Yaskawa INFORM job: aprem2TRJ1.JBI

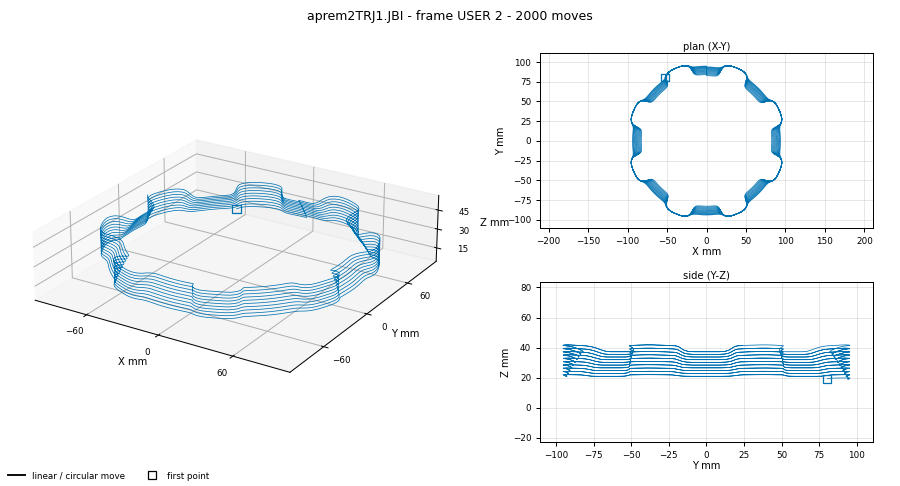
[picture p0: tool path of aprem2TRJ1.JBI in frame USER 2, 2000 of 2000 moves have a stored position in this frame; points joined in program order, loops and branches not executed]
/JOB
//NAME aprem2TRJ1
//POS
///NPOS 2000,0,2000,0,0,0
///USER 2
///TOOL 1
///POSTYPE USER
///RECTAN
///RCONF 1,0,0,0,0,0,0,0,0,0,0,0,0,0,0,0,0,0,0,0,0,0,0,0
C00000=-52.755,80.388,19.309,-171.7434,14.7955,0.0000
C00001=-51.961,81.931,19.493,-175.4363,10.0997,0.0000
C00002=-51.163,83.502,19.627,-176.4604,6.1368,0.0000
C00003=-49.917,85.194,19.692,-177.1673,3.1412,0.0000
C00004=-47.874,87.106,19.726,-178.6253,1.1228,0.0000
C00005=-45.272,88.975,19.753,-179.7684,0.1462,0.0000
C00006=-42.449,90.515,19.780,-179.9313,0.0331,0.0000
C00007=-39.659,91.796,19.798,-179.9923,0.0034,0.0000
C00008=-36.867,92.953,19.798,-179.9922,0.0031,0.0000
C00009=-33.988,94.020,19.780,-179.9280,0.0252,0.0000
C00010=-30.903,94.927,19.753,-179.7329,0.0604,0.0000
C00011=-27.741,95.446,19.726,-178.2343,0.1783,0.0000
C00012=-24.945,95.538,19.692,-175.7796,-0.2187,0.0000
C00013=-22.867,95.222,19.627,-173.1704,-1.8493,0.0000
C00014=-21.192,94.676,19.493,-169.6633,-3.9762,0.0000
C00015=-19.540,94.146,19.309,-163.8609,-4.8105,0.0000
C00016=-17.528,93.824,19.120,-157.6135,-2.4711,0.0000
C00017=-14.592,93.857,18.976,-154.0584,1.6115,0.0000
C00018=-10.190,94.262,18.917,-153.0799,2.7335,0.0000
C00019=-5.317,94.652,18.914,-152.9496,1.6756,0.0000
C00020=0.000,94.804,18.916,-152.9230,0.0002,0.0000
C00021=0.000,93.772,20.859,-151.1709,0.0003,0.0000
C00022=5.223,93.624,20.857,-151.1986,-1.7982,0.0000
C00023=10.031,93.243,20.860,-151.3318,-2.8339,0.0000
C00024=14.399,92.874,20.935,-152.4025,-1.1034,0.0000
C00025=17.292,92.935,21.118,-156.8210,4.1648,0.0000
C00026=19.271,93.399,21.361,-164.4264,6.3648,0.0000
C00027=20.902,94.108,21.598,-170.7334,4.7910,0.0000
C00028=22.556,94.852,21.773,-173.9772,2.3273,0.0000
C00029=24.607,95.353,21.858,-176.1452,0.4720,0.0000
C00030=27.423,95.407,21.902,-178.4246,-0.0969,0.0000
C00031=30.651,94.973,21.938,-179.8436,-0.0322,0.0000
C00032=33.828,94.073,21.973,-179.9356,-0.0223,0.0000
C00033=36.813,92.974,21.997,-179.9932,-0.0027,0.0000
C00034=39.712,91.773,21.997,-179.9933,-0.0029,0.0000
C00035=42.599,90.440,21.973,-179.9387,-0.0298,0.0000
C00036=45.483,88.829,21.938,-179.8667,-0.0878,0.0000
C00037=48.072,86.854,21.902,-178.8174,-1.0456,0.0000
C00038=50.025,84.825,21.858,-177.6053,-3.0607,0.0000
C00039=51.121,83.020,21.773,-177.3739,-5.9001,0.0000
C00040=51.765,81.324,21.598,-176.7889,-9.9060,0.0000
C00041=52.416,79.670,21.361,-173.2589,-15.4269,0.0000
C00042=53.488,77.942,21.118,-165.8953,-19.5067,0.0000
C00043=55.491,75.854,20.935,-159.0309,-19.5961,0.0000
C00044=58.840,73.026,20.860,-157.1386,-19.3725,0.0000
C00045=62.509,69.895,20.857,-157.6594,-20.1308,0.0000
C00046=66.307,66.307,20.859,-158.7340,-21.2663,0.0000
C00047=69.895,62.509,20.857,-159.8689,-22.3404,0.0000
C00048=73.026,58.840,20.860,-160.6271,-22.8610,0.0000
C00049=75.854,55.491,20.935,-160.4041,-20.9693,0.0000
C00050=77.942,53.488,21.118,-160.4933,-14.1047,0.0000
C00051=79.670,52.416,21.361,-164.5731,-6.7411,0.0000
C00052=81.324,51.765,21.598,-170.0940,-3.2111,0.0000
C00053=83.020,51.121,21.773,-174.0999,-2.6261,0.0000
C00054=84.825,50.025,21.858,-176.9393,-2.3947,0.0000
C00055=86.854,48.072,21.902,-178.9544,-1.1826,0.0000
C00056=88.829,45.483,21.938,-179.9122,-0.1333,0.0000
C00057=90.440,42.599,21.973,-179.9702,-0.0613,0.0000
C00058=91.773,39.712,21.997,-179.9971,-0.0067,0.0000
C00059=92.974,36.813,21.997,-179.9973,-0.0068,0.0000
C00060=94.073,33.828,21.973,-179.9777,-0.0644,0.0000
C00061=94.973,30.651,21.938,-179.9678,-0.1564,0.0000
C00062=95.407,27.423,21.902,-179.9031,-1.5754,0.0000
C00063=95.353,24.607,21.858,179.5280,-3.8548,0.0000
C00064=94.852,22.556,21.773,177.6727,-6.0228,0.0000
C00065=94.108,20.902,21.598,175.2090,-9.2666,0.0000
C00066=93.399,19.271,21.361,173.6352,-15.5736,0.0000
C00067=92.935,17.292,21.118,175.8352,-23.1790,0.0000
C00068=92.874,14.399,20.935,-178.8966,-27.5975,0.0000
C00069=93.243,10.031,20.860,-177.1661,-28.6682,0.0000
C00070=93.624,5.223,20.857,-178.2018,-28.8014,0.0000
C00071=93.772,0.000,20.859,179.9997,-28.8291,0.0000
C00072=93.624,-5.223,20.857,178.2021,-28.8014,0.0000
C00073=93.243,-10.031,20.860,177.1667,-28.6682,0.0000
C00074=92.875,-14.399,20.935,178.8963,-27.5974,0.0000
C00075=92.935,-17.292,21.118,-175.8352,-23.1790,0.0000
C00076=93.399,-19.271,21.361,-173.6352,-15.5736,0.0000
C00077=94.108,-20.902,21.598,-175.2090,-9.2666,0.0000
C00078=94.852,-22.556,21.773,-177.6727,-6.0228,0.0000
C00079=95.353,-24.607,21.858,-179.5280,-3.8548,0.0000
C00080=95.407,-27.423,21.902,179.9031,-1.5754,0.0000
C00081=94.973,-30.651,21.938,179.9678,-0.1564,0.0000
C00082=94.073,-33.828,21.973,179.9777,-0.0644,0.0000
C00083=92.974,-36.813,21.997,179.9973,-0.0068,0.0000
C00084=91.773,-39.712,21.997,179.9971,-0.0067,0.0000
C00085=90.440,-42.599,21.973,179.9702,-0.0613,0.0000
C00086=88.829,-45.483,21.938,179.9122,-0.1333,0.0000
C00087=86.854,-48.072,21.902,178.9544,-1.1826,0.0000
C00088=84.825,-50.025,21.858,176.9393,-2.3947,0.0000
C00089=83.020,-51.121,21.773,174.0999,-2.6261,0.0000
C00090=81.324,-51.765,21.598,170.0940,-3.2111,0.0000
C00091=79.670,-52.416,21.361,164.5731,-6.7411,0.0000
C00092=77.942,-53.488,21.118,160.4933,-14.1047,0.0000
C00093=75.854,-55.491,20.935,160.4039,-20.9691,0.0000
C00094=73.026,-58.840,20.860,160.6275,-22.8614,0.0000
C00095=69.895,-62.509,20.857,159.8692,-22.3406,0.0000
C00096=66.307,-66.307,20.859,158.7337,-21.2660,0.0000
C00097=62.509,-69.895,20.857,157.6596,-20.1311,0.0000
C00098=58.840,-73.026,20.860,157.1390,-19.3729,0.0000
C00099=55.491,-75.854,20.935,159.0307,-19.5959,0.0000
C00100=53.488,-77.942,21.118,165.8953,-19.5067,0.0000
C00101=52.416,-79.670,21.361,173.2589,-15.4269,0.0000
C00102=51.765,-81.324,21.598,176.7889,-9.9060,0.0000
C00103=51.121,-83.020,21.773,177.3739,-5.9001,0.0000
C00104=50.025,-84.825,21.858,177.6053,-3.0607,0.0000
C00105=48.072,-86.854,21.902,178.8174,-1.0456,0.0000
C00106=45.483,-88.829,21.938,179.8667,-0.0878,0.0000
C00107=42.599,-90.440,21.973,179.9387,-0.0298,0.0000
C00108=39.712,-91.773,21.997,179.9933,-0.0029,0.0000
C00109=36.813,-92.974,21.997,179.9932,-0.0027,0.0000
C00110=33.828,-94.073,21.973,179.9356,-0.0223,0.0000
C00111=30.651,-94.973,21.938,179.8436,-0.0322,0.0000
C00112=27.423,-95.407,21.902,178.4246,-0.0969,0.0000
C00113=24.607,-95.353,21.858,176.1452,0.4720,0.0000
C00114=22.556,-94.852,21.773,173.9772,2.3273,0.0000
C00115=20.902,-94.108,21.598,170.7334,4.7910,0.0000
C00116=19.271,-93.399,21.361,164.4264,6.3648,0.0000
C00117=17.292,-92.935,21.118,156.8210,4.1648,0.0000
C00118=14.399,-92.874,20.935,152.4025,-1.1034,0.0000
C00119=10.031,-93.243,20.860,151.3318,-2.8339,0.0000
C00120=5.223,-93.624,20.857,151.1986,-1.7982,0.0000
C00121=0.000,-93.772,20.859,151.1709,0.0003,0.0000
C00122=0.000,-93.772,20.859,151.1709,0.0003,0.0000
C00123=-5.223,-93.624,20.857,151.1986,1.7979,0.0000
C00124=-10.031,-93.243,20.860,151.3318,2.8333,0.0000
C00125=-14.399,-92.875,20.935,152.4026,1.1037,0.0000
C00126=-17.292,-92.935,21.118,156.8210,-4.1648,0.0000
C00127=-19.271,-93.399,21.361,164.4264,-6.3648,0.0000
C00128=-20.902,-94.108,21.598,170.7334,-4.7910,0.0000
C00129=-22.556,-94.852,21.773,173.9772,-2.3273,0.0000
C00130=-24.607,-95.353,21.858,176.1452,-0.4720,0.0000
C00131=-27.423,-95.407,21.902,178.4246,0.0969,0.0000
C00132=-30.651,-94.973,21.938,179.8436,0.0322,0.0000
C00133=-33.828,-94.073,21.973,179.9356,0.0223,0.0000
C00134=-36.813,-92.974,21.997,179.9932,0.0027,0.0000
C00135=-39.712,-91.773,21.997,179.9933,0.0029,0.0000
C00136=-42.599,-90.440,21.973,179.9387,0.0298,0.0000
C00137=-45.483,-88.829,21.938,179.8667,0.0878,0.0000
C00138=-48.072,-86.854,21.902,178.8174,1.0456,0.0000
C00139=-50.025,-84.825,21.858,177.6053,3.0607,0.0000
C00140=-51.121,-83.020,21.773,177.3739,5.9001,0.0000
C00141=-51.765,-81.324,21.598,176.7889,9.9060,0.0000
C00142=-52.416,-79.670,21.361,173.2589,15.4269,0.0000
C00143=-53.488,-77.942,21.118,165.8953,19.5067,0.0000
C00144=-55.491,-75.854,20.935,159.0309,19.5961,0.0000
C00145=-58.840,-73.026,20.860,157.1386,19.3725,0.0000
C00146=-62.509,-69.895,20.857,157.6594,20.1308,0.0000
C00147=-66.307,-66.307,20.859,158.7340,21.2663,0.0000
C00148=-69.895,-62.509,20.857,159.8689,22.3404,0.0000
C00149=-73.026,-58.840,20.860,160.6271,22.8610,0.0000
C00150=-75.854,-55.491,20.935,160.4041,20.9693,0.0000
C00151=-77.942,-53.488,21.118,160.4933,14.1047,0.0000
C00152=-79.670,-52.416,21.361,164.5731,6.7411,0.0000
C00153=-81.324,-51.765,21.598,170.0940,3.2111,0.0000
C00154=-83.020,-51.121,21.773,174.0999,2.6261,0.0000
C00155=-84.825,-50.025,21.858,176.9393,2.3947,0.0000
C00156=-86.854,-48.072,21.902,178.9544,1.1826,0.0000
C00157=-88.829,-45.483,21.938,179.9122,0.1333,0.0000
C00158=-90.440,-42.599,21.973,179.9702,0.0613,0.0000
C00159=-91.773,-39.712,21.997,179.9971,0.0067,0.0000
C00160=-92.974,-36.813,21.997,179.9973,0.0068,0.0000
C00161=-94.073,-33.828,21.973,179.9777,0.0644,0.0000
C00162=-94.973,-30.651,21.938,179.9678,0.1564,0.0000
C00163=-95.407,-27.423,21.902,179.9031,1.5754,0.0000
C00164=-95.353,-24.607,21.858,-179.5280,3.8548,0.0000
C00165=-94.852,-22.556,21.773,-177.6727,6.0228,0.0000
C00166=-94.108,-20.902,21.598,-175.2090,9.2666,0.0000
C00167=-93.399,-19.271,21.361,-173.6352,15.5736,0.0000
C00168=-92.935,-17.292,21.118,-175.8352,23.1790,0.0000
C00169=-92.874,-14.399,20.935,178.8966,27.5975,0.0000
C00170=-93.243,-10.031,20.860,177.1661,28.6682,0.0000
C00171=-93.624,-5.223,20.857,178.2018,28.8014,0.0000
C00172=-93.772,0.000,20.859,-179.9997,28.8291,0.0000
C00173=-93.624,5.223,20.857,-178.2021,28.8014,0.0000
C00174=-93.243,10.031,20.860,-177.1667,28.6682,0.0000
C00175=-92.875,14.399,20.935,-178.8963,27.5974,0.0000
C00176=-92.935,17.292,21.118,175.8352,23.1790,0.0000
C00177=-93.399,19.271,21.361,173.6352,15.5736,0.0000
C00178=-94.108,20.902,21.598,175.2090,9.2666,0.0000
C00179=-94.852,22.556,21.773,177.6727,6.0228,0.0000
C00180=-95.353,24.607,21.858,179.5280,3.8548,0.0000
C00181=-95.407,27.423,21.902,-179.9031,1.5754,0.0000
C00182=-94.973,30.651,21.938,-179.9678,0.1564,0.0000
C00183=-94.073,33.828,21.973,-179.9777,0.0644,0.0000
C00184=-92.974,36.813,21.997,-179.9973,0.0068,0.0000
C00185=-91.773,39.712,21.997,-179.9971,0.0067,0.0000
C00186=-90.440,42.599,21.973,-179.9702,0.0613,0.0000
C00187=-88.829,45.483,21.938,-179.9122,0.1333,0.0000
C00188=-86.854,48.072,21.902,-178.9544,1.1826,0.0000
C00189=-84.825,50.025,21.858,-176.9393,2.3947,0.0000
C00190=-83.020,51.121,21.773,-174.0999,2.6261,0.0000
C00191=-81.324,51.765,21.598,-170.0940,3.2111,0.0000
C00192=-79.670,52.416,21.361,-164.5731,6.7411,0.0000
C00193=-77.942,53.488,21.118,-160.4933,14.1047,0.0000
C00194=-75.854,55.491,20.935,-160.4039,20.9691,0.0000
C00195=-73.026,58.840,20.860,-160.6275,22.8614,0.0000
C00196=-69.895,62.509,20.857,-159.8692,22.3406,0.0000
C00197=-66.307,66.307,20.859,-158.7337,21.2660,0.0000
C00198=-62.509,69.895,20.857,-157.6596,20.1311,0.0000
C00199=-58.840,73.026,20.860,-157.1390,19.3729,0.0000
C00200=-55.491,75.854,20.935,-159.0307,19.5959,0.0000
C00201=-53.488,77.942,21.118,-165.8953,19.5067,0.0000
C00202=-52.416,79.670,21.361,-173.2589,15.4269,0.0000
C00203=-51.765,81.324,21.598,-176.7889,9.9060,0.0000
C00204=-51.121,83.020,21.773,-177.3739,5.9001,0.0000
C00205=-50.025,84.825,21.858,-177.6053,3.0607,0.0000
C00206=-48.072,86.854,21.902,-178.8174,1.0456,0.0000
C00207=-45.483,88.829,21.938,-179.8667,0.0878,0.0000
C00208=-42.599,90.440,21.973,-179.9387,0.0298,0.0000
C00209=-39.712,91.773,21.997,-179.9933,0.0029,0.0000
C00210=-36.813,92.974,21.997,-179.9932,0.0027,0.0000
C00211=-33.828,94.073,21.973,-179.9356,0.0223,0.0000
C00212=-30.651,94.973,21.938,-179.8436,0.0322,0.0000
C00213=-27.423,95.407,21.902,-178.4246,0.0969,0.0000
C00214=-24.607,95.353,21.858,-176.1452,-0.4720,0.0000
C00215=-22.556,94.852,21.773,-173.9772,-2.3273,0.0000
C00216=-20.902,94.108,21.598,-170.7334,-4.7910,0.0000
C00217=-19.271,93.399,21.361,-164.4264,-6.3648,0.0000
C00218=-17.292,92.935,21.118,-156.8210,-4.1648,0.0000
C00219=-14.399,92.875,20.935,-152.4026,1.1037,0.0000
C00220=-10.031,93.243,20.860,-151.3318,2.8333,0.0000
C00221=-5.223,93.624,20.857,-151.1986,1.7979,0.0000
C00222=0.000,93.772,20.859,-151.1709,0.0003,0.0000
C00223=0.000,92.684,22.771,-149.6099,0.0003,0.0000
C00224=5.124,92.540,22.769,-149.6384,-1.9089,0.0000
C00225=9.864,92.169,22.773,-149.7740,-2.8935,0.0000
C00226=14.194,91.838,22.865,-150.9609,-0.4562,0.0000
C00227=17.042,91.994,23.091,-156.4950,5.9927,0.0000
C00228=18.986,92.606,23.393,-165.5257,7.6266,0.0000
C00229=20.592,93.503,23.691,-172.1237,5.1935,0.0000
C00230=22.223,94.456,23.912,-175.0607,2.5303,0.0000
C00231=24.245,95.156,24.019,-176.7061,0.6541,0.0000
C00232=27.082,95.366,24.075,-178.6926,-0.0269,0.0000
C00233=30.380,95.022,24.120,-179.9786,-0.0040,0.0000
C00234=33.658,94.129,24.166,-179.9455,-0.0187,0.0000
C00235=36.755,92.996,24.196,-179.9945,-0.0022,0.0000
C00236=39.769,91.748,24.196,-179.9946,-0.0024,0.0000
C00237=42.760,90.359,24.166,-179.9482,-0.0253,0.0000
C00238=45.709,88.673,24.120,-179.9821,-0.0123,0.0000
C00239=48.284,86.584,24.075,-179.0565,-0.9056,0.0000
C00240=50.142,84.429,24.019,-178.1315,-2.7920,0.0000
C00241=51.076,82.504,23.912,-178.2896,-5.2767,0.0000
C00242=51.556,80.678,23.691,-178.0785,-9.2071,0.0000
C00243=52.057,78.907,23.393,-174.9794,-15.4942,0.0000
C00244=52.999,77.101,23.091,-166.8676,-20.8949,0.0000
C00245=54.903,74.976,22.865,-158.2868,-21.1542,0.0000
C00246=58.198,72.148,22.773,-155.8812,-20.6181,0.0000
C00247=61.813,69.059,22.769,-156.3569,-21.3383,0.0000
C00248=65.538,65.538,22.771,-157.4767,-22.5237,0.0000
C00249=69.059,61.813,22.769,-158.6615,-23.6429,0.0000
C00250=72.148,58.198,22.773,-159.3815,-24.1184,0.0000
C00251=74.976,54.903,22.865,-158.8460,-21.7135,0.0000
C00252=77.101,52.999,23.091,-159.1051,-13.1324,0.0000
C00253=78.907,52.057,23.393,-164.5058,-5.0206,0.0000
C00254=80.678,51.556,23.691,-170.7929,-1.9215,0.0000
C00255=82.504,51.076,23.912,-174.7233,-1.7104,0.0000
C00256=84.429,50.142,24.019,-177.2080,-1.8685,0.0000
C00257=86.584,48.284,24.075,-179.0944,-0.9435,0.0000
C00258=88.673,45.709,24.120,-179.9877,-0.0179,0.0000
C00259=90.359,42.760,24.166,-179.9747,-0.0518,0.0000
C00260=91.748,39.769,24.196,-179.9976,-0.0054,0.0000
C00261=92.996,36.755,24.196,-179.9978,-0.0055,0.0000
C00262=94.129,33.658,24.166,-179.9813,-0.0545,0.0000
C00263=95.022,30.380,24.120,-179.9960,-0.0214,0.0000
C00264=95.366,27.082,24.075,-179.9731,-1.3074,0.0000
C00265=95.156,24.245,24.019,179.3459,-3.2939,0.0000
C00266=94.456,22.223,23.912,177.4697,-4.9393,0.0000
C00267=93.503,20.592,23.691,174.8065,-7.8763,0.0000
C00268=92.606,18.986,23.393,172.3734,-14.4743,0.0000
C00269=91.994,17.042,23.091,174.0073,-23.5050,0.0000
C00270=91.838,14.194,22.865,-179.5438,-29.0391,0.0000
C00271=92.169,9.864,22.773,-177.1065,-30.2260,0.0000
C00272=92.540,5.124,22.769,-178.0911,-30.3616,0.0000
C00273=92.684,0.000,22.771,179.9997,-30.3901,0.0000
C00274=92.540,-5.124,22.769,178.0916,-30.3616,0.0000
C00275=92.169,-9.864,22.773,177.1071,-30.2260,0.0000
C00276=91.838,-14.194,22.865,179.5434,-29.0390,0.0000
C00277=91.994,-17.042,23.091,-174.0073,-23.5050,0.0000
C00278=92.606,-18.986,23.393,-172.3734,-14.4743,0.0000
C00279=93.503,-20.592,23.691,-174.8065,-7.8763,0.0000
C00280=94.456,-22.223,23.912,-177.4697,-4.9393,0.0000
C00281=95.156,-24.245,24.019,-179.3459,-3.2939,0.0000
C00282=95.366,-27.082,24.075,179.9731,-1.3074,0.0000
C00283=95.022,-30.380,24.120,179.9960,-0.0214,0.0000
C00284=94.129,-33.658,24.166,179.9813,-0.0545,0.0000
C00285=92.996,-36.755,24.196,179.9978,-0.0055,0.0000
C00286=91.748,-39.769,24.196,179.9976,-0.0054,0.0000
C00287=90.359,-42.760,24.166,179.9747,-0.0518,0.0000
C00288=88.673,-45.709,24.120,179.9877,-0.0179,0.0000
C00289=86.584,-48.284,24.075,179.0944,-0.9435,0.0000
C00290=84.429,-50.142,24.019,177.2080,-1.8685,0.0000
C00291=82.504,-51.076,23.912,174.7233,-1.7104,0.0000
C00292=80.678,-51.556,23.691,170.7929,-1.9215,0.0000
C00293=78.907,-52.057,23.393,164.5058,-5.0206,0.0000
C00294=77.101,-52.999,23.091,159.1051,-13.1324,0.0000
C00295=74.976,-54.903,22.865,158.8458,-21.7132,0.0000
C00296=72.148,-58.198,22.773,159.3819,-24.1188,0.0000
C00297=69.059,-61.813,22.769,158.6617,-23.6431,0.0000
C00298=65.538,-65.538,22.771,157.4763,-22.5233,0.0000
C00299=61.813,-69.059,22.769,156.3571,-21.3385,0.0000
C00300=58.198,-72.148,22.773,155.8816,-20.6185,0.0000
C00301=54.903,-74.976,22.865,158.2865,-21.1540,0.0000
C00302=52.999,-77.101,23.091,166.8676,-20.8949,0.0000
C00303=52.057,-78.907,23.393,174.9794,-15.4942,0.0000
C00304=51.556,-80.678,23.691,178.0785,-9.2071,0.0000
C00305=51.076,-82.504,23.912,178.2896,-5.2767,0.0000
C00306=50.142,-84.429,24.019,178.1315,-2.7920,0.0000
C00307=48.284,-86.584,24.075,179.0565,-0.9056,0.0000
C00308=45.709,-88.673,24.120,179.9821,-0.0123,0.0000
C00309=42.760,-90.359,24.166,179.9482,-0.0253,0.0000
C00310=39.769,-91.748,24.196,179.9946,-0.0024,0.0000
C00311=36.755,-92.996,24.196,179.9945,-0.0022,0.0000
C00312=33.658,-94.129,24.166,179.9455,-0.0187,0.0000
C00313=30.380,-95.022,24.120,179.9786,-0.0040,0.0000
C00314=27.082,-95.366,24.075,178.6926,-0.0269,0.0000
C00315=24.245,-95.156,24.019,176.7061,0.6541,0.0000
C00316=22.223,-94.456,23.912,175.0607,2.5303,0.0000
C00317=20.592,-93.503,23.691,172.1237,5.1935,0.0000
C00318=18.986,-92.606,23.393,165.5257,7.6266,0.0000
C00319=17.042,-91.994,23.091,156.4950,5.9927,0.0000
C00320=14.194,-91.838,22.865,150.9609,-0.4562,0.0000
C00321=9.864,-92.169,22.773,149.7740,-2.8935,0.0000
C00322=5.124,-92.540,22.769,149.6384,-1.9089,0.0000
C00323=0.000,-92.684,22.771,149.6099,0.0003,0.0000
C00324=0.000,-92.684,22.771,149.6099,0.0003,0.0000
C00325=-5.124,-92.540,22.769,149.6384,1.9084,0.0000
C00326=-9.864,-92.169,22.773,149.7740,2.8929,0.0000
C00327=-14.194,-91.838,22.865,150.9610,0.4566,0.0000
C00328=-17.042,-91.994,23.091,156.4950,-5.9927,0.0000
C00329=-18.986,-92.606,23.393,165.5257,-7.6266,0.0000
C00330=-20.592,-93.503,23.691,172.1237,-5.1935,0.0000
C00331=-22.223,-94.456,23.912,175.0607,-2.5303,0.0000
C00332=-24.245,-95.156,24.019,176.7061,-0.6541,0.0000
C00333=-27.082,-95.366,24.075,178.6926,0.0269,0.0000
C00334=-30.380,-95.022,24.120,179.9786,0.0040,0.0000
C00335=-33.658,-94.129,24.166,179.9455,0.0187,0.0000
C00336=-36.755,-92.996,24.196,179.9945,0.0022,0.0000
C00337=-39.769,-91.748,24.196,179.9946,0.0024,0.0000
C00338=-42.760,-90.359,24.166,179.9482,0.0253,0.0000
C00339=-45.709,-88.673,24.120,179.9821,0.0123,0.0000
C00340=-48.284,-86.584,24.075,179.0565,0.9056,0.0000
C00341=-50.142,-84.429,24.019,178.1315,2.7920,0.0000
C00342=-51.076,-82.504,23.912,178.2896,5.2767,0.0000
C00343=-51.556,-80.678,23.691,178.0785,9.2071,0.0000
C00344=-52.057,-78.907,23.393,174.9794,15.4942,0.0000
C00345=-52.999,-77.101,23.091,166.8676,20.8949,0.0000
C00346=-54.903,-74.976,22.865,158.2868,21.1542,0.0000
C00347=-58.198,-72.148,22.773,155.8812,20.6181,0.0000
C00348=-61.813,-69.059,22.769,156.3569,21.3383,0.0000
C00349=-65.538,-65.538,22.771,157.4767,22.5237,0.0000
C00350=-69.059,-61.813,22.769,158.6615,23.6429,0.0000
C00351=-72.148,-58.198,22.773,159.3815,24.1184,0.0000
C00352=-74.976,-54.903,22.865,158.8460,21.7135,0.0000
C00353=-77.101,-52.999,23.091,159.1051,13.1324,0.0000
C00354=-78.907,-52.057,23.393,164.5058,5.0206,0.0000
C00355=-80.678,-51.556,23.691,170.7929,1.9215,0.0000
C00356=-82.504,-51.076,23.912,174.7233,1.7104,0.0000
C00357=-84.429,-50.142,24.019,177.2080,1.8685,0.0000
C00358=-86.584,-48.284,24.075,179.0944,0.9435,0.0000
C00359=-88.673,-45.709,24.120,179.9877,0.0179,0.0000
C00360=-90.359,-42.760,24.166,179.9747,0.0518,0.0000
C00361=-91.748,-39.769,24.196,179.9976,0.0054,0.0000
C00362=-92.996,-36.755,24.196,179.9978,0.0055,0.0000
C00363=-94.129,-33.658,24.166,179.9813,0.0545,0.0000
C00364=-95.022,-30.380,24.120,179.9960,0.0214,0.0000
C00365=-95.366,-27.082,24.075,179.9731,1.3074,0.0000
C00366=-95.156,-24.245,24.019,-179.3459,3.2939,0.0000
C00367=-94.456,-22.223,23.912,-177.4697,4.9393,0.0000
C00368=-93.503,-20.592,23.691,-174.8065,7.8763,0.0000
C00369=-92.606,-18.986,23.393,-172.3734,14.4743,0.0000
C00370=-91.994,-17.042,23.091,-174.0073,23.5050,0.0000
C00371=-91.838,-14.194,22.865,179.5438,29.0391,0.0000
C00372=-92.169,-9.864,22.773,177.1065,30.2260,0.0000
C00373=-92.540,-5.124,22.769,178.0911,30.3616,0.0000
C00374=-92.684,0.000,22.771,-179.9997,30.3901,0.0000
C00375=-92.540,5.124,22.769,-178.0916,30.3616,0.0000
C00376=-92.169,9.864,22.773,-177.1071,30.2260,0.0000
C00377=-91.838,14.194,22.865,-179.5434,29.0390,0.0000
C00378=-91.994,17.042,23.091,174.0073,23.5050,0.0000
C00379=-92.606,18.986,23.393,172.3734,14.4743,0.0000
C00380=-93.503,20.592,23.691,174.8065,7.8763,0.0000
C00381=-94.456,22.223,23.912,177.4697,4.9393,0.0000
C00382=-95.156,24.245,24.019,179.3459,3.2939,0.0000
C00383=-95.366,27.082,24.075,-179.9731,1.3074,0.0000
C00384=-95.022,30.380,24.120,-179.9960,0.0214,0.0000
C00385=-94.129,33.658,24.166,-179.9813,0.0545,0.0000
C00386=-92.996,36.755,24.196,-179.9978,0.0055,0.0000
C00387=-91.748,39.769,24.196,-179.9976,0.0054,0.0000
C00388=-90.359,42.760,24.166,-179.9747,0.0518,0.0000
C00389=-88.673,45.709,24.120,-179.9877,0.0179,0.0000
C00390=-86.584,48.284,24.075,-179.0944,0.9435,0.0000
C00391=-84.429,50.142,24.019,-177.2080,1.8685,0.0000
C00392=-82.504,51.076,23.912,-174.7233,1.7104,0.0000
C00393=-80.678,51.556,23.691,-170.7929,1.9215,0.0000
C00394=-78.907,52.057,23.393,-164.5058,5.0206,0.0000
C00395=-77.101,52.999,23.091,-159.1051,13.1324,0.0000
C00396=-74.976,54.903,22.865,-158.8458,21.7132,0.0000
C00397=-72.148,58.198,22.773,-159.3819,24.1188,0.0000
C00398=-69.059,61.813,22.769,-158.6617,23.6431,0.0000
C00399=-65.538,65.538,22.771,-157.4763,22.5233,0.0000
C00400=-61.813,69.059,22.769,-156.3571,21.3385,0.0000
C00401=-58.198,72.148,22.773,-155.8816,20.6185,0.0000
C00402=-54.903,74.976,22.865,-158.2865,21.1540,0.0000
C00403=-52.999,77.101,23.091,-166.8676,20.8949,0.0000
C00404=-52.057,78.907,23.393,-174.9794,15.4942,0.0000
C00405=-51.556,80.678,23.691,-178.0785,9.2071,0.0000
C00406=-51.076,82.504,23.912,-178.2896,5.2767,0.0000
C00407=-50.142,84.429,24.019,-178.1315,2.7920,0.0000
C00408=-48.284,86.584,24.075,-179.0565,0.9056,0.0000
C00409=-45.709,88.673,24.120,-179.9821,0.0123,0.0000
C00410=-42.760,90.359,24.166,-179.9482,0.0253,0.0000
C00411=-39.769,91.748,24.196,-179.9946,0.0024,0.0000
C00412=-36.755,92.996,24.196,-179.9945,0.0022,0.0000
C00413=-33.658,94.129,24.166,-179.9455,0.0187,0.0000
C00414=-30.380,95.022,24.120,-179.9786,0.0040,0.0000
C00415=-27.082,95.366,24.075,-178.6926,0.0269,0.0000
C00416=-24.245,95.156,24.019,-176.7061,-0.6541,0.0000
C00417=-22.223,94.456,23.912,-175.0607,-2.5303,0.0000
C00418=-20.592,93.503,23.691,-172.1237,-5.1935,0.0000
C00419=-18.986,92.606,23.393,-165.5257,-7.6266,0.0000
C00420=-17.042,91.994,23.091,-156.4950,-5.9927,0.0000
C00421=-14.194,91.838,22.865,-150.9610,0.4566,0.0000
C00422=-9.864,92.169,22.773,-149.7740,2.8929,0.0000
C00423=-5.124,92.540,22.769,-149.6384,1.9084,0.0000
C00424=0.000,92.684,22.771,-149.6099,0.0003,0.0000
C00425=0.000,91.548,24.655,-148.2220,0.0004,0.0000
C00426=5.020,91.408,24.652,-148.2512,-2.0082,0.0000
C00427=9.690,91.047,24.657,-148.3888,-2.9141,0.0000
C00428=13.981,90.755,24.767,-149.7234,0.3213,0.0000
C00429=16.781,91.008,25.041,-156.6468,7.8344,0.0000
C00430=18.686,91.772,25.406,-167.0189,8.4697,0.0000
C00431=20.265,92.865,25.771,-173.6442,5.1590,0.0000
C00432=21.871,94.037,26.043,-176.2884,2.4064,0.0000
C00433=23.861,94.948,26.175,-177.4309,0.7190,0.0000
C00434=26.720,95.323,26.245,-179.0289,0.0208,0.0000
C00435=30.093,95.074,26.301,179.8658,0.0220,0.0000
C00436=33.476,94.189,26.358,-179.9573,-0.0145,0.0000
C00437=36.693,93.020,26.395,-179.9960,-0.0016,0.0000
C00438=39.829,91.721,26.395,-179.9960,-0.0018,0.0000
C00439=42.931,90.273,26.358,-179.9596,-0.0199,0.0000
C00440=45.948,88.507,26.301,179.8895,0.0793,0.0000
C00441=48.509,86.297,26.245,-179.3280,-0.7014,0.0000
C00442=50.266,84.010,26.175,-178.6908,-2.3250,0.0000
C00443=51.029,81.959,26.043,-179.0745,-4.3225,0.0000
C00444=51.336,79.995,25.771,-179.1451,-8.1159,0.0000
C00445=51.679,78.105,25.406,-176.6973,-15.0186,0.0000
C00446=52.487,76.218,25.041,-168.2493,-21.9298,0.0000
C00447=54.287,74.059,24.767,-157.7629,-22.6253,0.0000
C00448=57.528,71.231,24.657,-154.7702,-21.7624,0.0000
C00449=61.085,68.184,24.652,-155.1868,-22.4287,0.0000
C00450=64.734,64.734,24.655,-156.3444,-23.6560,0.0000
C00451=68.184,61.085,24.652,-157.5710,-24.8129,0.0000
C00452=71.231,57.528,24.657,-158.2372,-25.2293,0.0000
C00453=74.059,54.287,24.767,-157.3750,-22.2374,0.0000
C00454=76.218,52.487,25.041,-158.0702,-11.7507,0.0000
C00455=78.105,51.679,25.406,-164.9814,-3.3027,0.0000
C00456=79.995,51.336,25.771,-171.8841,-0.8549,0.0000
C00457=81.959,51.029,26.043,-175.6775,-0.9255,0.0000
C00458=84.010,50.266,26.175,-177.6750,-1.3092,0.0000
C00459=86.297,48.509,26.245,-179.2986,-0.6720,0.0000
C00460=88.507,45.948,26.301,179.9207,0.1105,0.0000
C00461=90.273,42.931,26.358,-179.9801,-0.0404,0.0000
C00462=91.721,39.829,26.395,-179.9982,-0.0040,0.0000
C00463=93.020,36.693,26.395,-179.9984,-0.0040,0.0000
C00464=94.189,33.476,26.358,-179.9855,-0.0427,0.0000
C00465=95.074,30.093,26.301,179.9780,0.1342,0.0000
C00466=95.323,26.720,26.245,179.9792,-0.9711,0.0000
C00467=94.948,23.861,26.175,179.2810,-2.5691,0.0000
C00468=94.037,21.871,26.043,177.5936,-3.7116,0.0000
C00469=92.865,20.265,25.771,174.8410,-6.3558,0.0000
C00470=91.772,18.686,25.406,171.5303,-12.9811,0.0000
C00471=91.008,16.781,25.041,172.1656,-23.3532,0.0000
C00472=90.755,13.981,24.767,179.6787,-30.2766,0.0000
C00473=91.047,9.690,24.657,-177.0859,-31.6112,0.0000
C00474=91.408,5.020,24.652,-177.9918,-31.7488,0.0000
C00475=91.548,0.000,24.655,179.9996,-31.7780,0.0000
C00476=91.408,-5.020,24.652,177.9923,-31.7488,0.0000
C00477=91.047,-9.690,24.657,177.0867,-31.6111,0.0000
C00478=90.755,-13.981,24.767,-179.6793,-30.2766,0.0000
C00479=91.008,-16.781,25.041,-172.1656,-23.3532,0.0000
C00480=91.772,-18.686,25.406,-171.5303,-12.9811,0.0000
C00481=92.865,-20.265,25.771,-174.8410,-6.3558,0.0000
C00482=94.037,-21.871,26.043,-177.5936,-3.7116,0.0000
C00483=94.948,-23.861,26.175,-179.2810,-2.5691,0.0000
C00484=95.323,-26.720,26.245,-179.9792,-0.9711,0.0000
C00485=95.074,-30.093,26.301,-179.9780,0.1342,0.0000
C00486=94.189,-33.476,26.358,179.9855,-0.0427,0.0000
C00487=93.020,-36.693,26.395,179.9984,-0.0040,0.0000
C00488=91.721,-39.829,26.395,179.9982,-0.0040,0.0000
C00489=90.273,-42.931,26.358,179.9801,-0.0404,0.0000
C00490=88.507,-45.948,26.301,-179.9207,0.1105,0.0000
C00491=86.297,-48.509,26.245,179.2986,-0.6720,0.0000
C00492=84.010,-50.266,26.175,177.6750,-1.3092,0.0000
C00493=81.959,-51.029,26.043,175.6775,-0.9255,0.0000
C00494=79.995,-51.336,25.771,171.8841,-0.8549,0.0000
C00495=78.105,-51.679,25.406,164.9814,-3.3027,0.0000
C00496=76.218,-52.487,25.041,158.0702,-11.7507,0.0000
C00497=74.059,-54.287,24.767,157.3747,-22.2371,0.0000
C00498=71.231,-57.528,24.657,158.2376,-25.2298,0.0000
C00499=68.184,-61.085,24.652,157.5713,-24.8132,0.0000
C00500=64.734,-64.734,24.655,156.3440,-23.6556,0.0000
C00501=61.085,-68.184,24.652,155.1871,-22.4290,0.0000
C00502=57.528,-71.231,24.657,154.7707,-21.7628,0.0000
C00503=54.287,-74.059,24.767,157.7626,-22.6250,0.0000
C00504=52.487,-76.218,25.041,168.2493,-21.9298,0.0000
C00505=51.679,-78.105,25.406,176.6973,-15.0186,0.0000
C00506=51.336,-79.995,25.771,179.1451,-8.1159,0.0000
C00507=51.029,-81.959,26.043,179.0745,-4.3225,0.0000
C00508=50.266,-84.010,26.175,178.6908,-2.3250,0.0000
C00509=48.509,-86.297,26.245,179.3280,-0.7014,0.0000
C00510=45.948,-88.507,26.301,-179.8895,0.0793,0.0000
C00511=42.931,-90.273,26.358,179.9596,-0.0199,0.0000
C00512=39.829,-91.721,26.395,179.9960,-0.0018,0.0000
C00513=36.693,-93.020,26.395,179.9960,-0.0016,0.0000
C00514=33.476,-94.189,26.358,179.9573,-0.0145,0.0000
C00515=30.093,-95.074,26.301,-179.8658,0.0220,0.0000
C00516=26.720,-95.323,26.245,179.0289,0.0208,0.0000
C00517=23.861,-94.948,26.175,177.4309,0.7190,0.0000
C00518=21.871,-94.037,26.043,176.2884,2.4064,0.0000
C00519=20.265,-92.865,25.771,173.6442,5.1590,0.0000
C00520=18.686,-91.772,25.406,167.0189,8.4697,0.0000
C00521=16.781,-91.008,25.041,156.6468,7.8344,0.0000
C00522=13.981,-90.755,24.767,149.7234,0.3213,0.0000
C00523=9.690,-91.047,24.657,148.3888,-2.9141,0.0000
C00524=5.020,-91.408,24.652,148.2512,-2.0082,0.0000
C00525=0.000,-91.548,24.655,148.2220,0.0004,0.0000
C00526=0.000,-91.548,24.655,148.2220,0.0004,0.0000
C00527=-5.020,-91.408,24.652,148.2512,2.0077,0.0000
C00528=-9.690,-91.047,24.657,148.3889,2.9133,0.0000
C00529=-13.981,-90.755,24.767,149.7234,-0.3207,0.0000
C00530=-16.781,-91.008,25.041,156.6468,-7.8344,0.0000
C00531=-18.686,-91.772,25.406,167.0189,-8.4697,0.0000
C00532=-20.265,-92.865,25.771,173.6442,-5.1590,0.0000
C00533=-21.871,-94.037,26.043,176.2884,-2.4064,0.0000
C00534=-23.861,-94.948,26.175,177.4309,-0.7190,0.0000
C00535=-26.720,-95.323,26.245,179.0289,-0.0208,0.0000
C00536=-30.093,-95.074,26.301,-179.8658,-0.0220,0.0000
C00537=-33.476,-94.189,26.358,179.9573,0.0145,0.0000
C00538=-36.693,-93.020,26.395,179.9960,0.0016,0.0000
C00539=-39.829,-91.721,26.395,179.9960,0.0018,0.0000
C00540=-42.931,-90.273,26.358,179.9596,0.0199,0.0000
C00541=-45.948,-88.507,26.301,-179.8895,-0.0793,0.0000
C00542=-48.509,-86.297,26.245,179.3280,0.7014,0.0000
C00543=-50.266,-84.010,26.175,178.6908,2.3250,0.0000
C00544=-51.029,-81.959,26.043,179.0745,4.3225,0.0000
C00545=-51.336,-79.995,25.771,179.1451,8.1159,0.0000
C00546=-51.679,-78.105,25.406,176.6973,15.0186,0.0000
C00547=-52.487,-76.218,25.041,168.2493,21.9298,0.0000
C00548=-54.287,-74.059,24.767,157.7629,22.6253,0.0000
C00549=-57.528,-71.231,24.657,154.7702,21.7624,0.0000
C00550=-61.085,-68.184,24.652,155.1868,22.4287,0.0000
C00551=-64.734,-64.734,24.655,156.3444,23.6560,0.0000
C00552=-68.184,-61.085,24.652,157.5710,24.8129,0.0000
C00553=-71.231,-57.528,24.657,158.2372,25.2293,0.0000
C00554=-74.059,-54.287,24.767,157.3750,22.2374,0.0000
C00555=-76.218,-52.487,25.041,158.0702,11.7507,0.0000
C00556=-78.105,-51.679,25.406,164.9814,3.3027,0.0000
C00557=-79.995,-51.336,25.771,171.8841,0.8549,0.0000
C00558=-81.959,-51.029,26.043,175.6775,0.9255,0.0000
C00559=-84.010,-50.266,26.175,177.6750,1.3092,0.0000
C00560=-86.297,-48.509,26.245,179.2986,0.6720,0.0000
C00561=-88.507,-45.948,26.301,-179.9207,-0.1105,0.0000
C00562=-90.273,-42.931,26.358,179.9801,0.0404,0.0000
C00563=-91.721,-39.829,26.395,179.9982,0.0040,0.0000
C00564=-93.020,-36.693,26.395,179.9984,0.0040,0.0000
C00565=-94.189,-33.476,26.358,179.9855,0.0427,0.0000
C00566=-95.074,-30.093,26.301,-179.9780,-0.1342,0.0000
C00567=-95.323,-26.720,26.245,-179.9792,0.9711,0.0000
C00568=-94.948,-23.861,26.175,-179.2810,2.5691,0.0000
C00569=-94.037,-21.871,26.043,-177.5936,3.7116,0.0000
C00570=-92.865,-20.265,25.771,-174.8410,6.3558,0.0000
C00571=-91.772,-18.686,25.406,-171.5303,12.9811,0.0000
C00572=-91.008,-16.781,25.041,-172.1656,23.3532,0.0000
C00573=-90.755,-13.981,24.767,-179.6787,30.2766,0.0000
C00574=-91.047,-9.690,24.657,177.0859,31.6112,0.0000
C00575=-91.408,-5.020,24.652,177.9918,31.7488,0.0000
C00576=-91.548,0.000,24.655,-179.9996,31.7780,0.0000
C00577=-91.408,5.020,24.652,-177.9923,31.7488,0.0000
C00578=-91.047,9.690,24.657,-177.0867,31.6111,0.0000
C00579=-90.755,13.981,24.767,179.6793,30.2766,0.0000
C00580=-91.008,16.781,25.041,172.1656,23.3532,0.0000
C00581=-91.772,18.686,25.406,171.5303,12.9811,0.0000
C00582=-92.865,20.265,25.771,174.8410,6.3558,0.0000
C00583=-94.037,21.871,26.043,177.5936,3.7116,0.0000
C00584=-94.948,23.861,26.175,179.2810,2.5691,0.0000
C00585=-95.323,26.720,26.245,179.9792,0.9711,0.0000
C00586=-95.074,30.093,26.301,179.9780,-0.1342,0.0000
C00587=-94.189,33.476,26.358,-179.9855,0.0427,0.0000
C00588=-93.020,36.693,26.395,-179.9984,0.0040,0.0000
C00589=-91.721,39.829,26.395,-179.9982,0.0040,0.0000
C00590=-90.273,42.931,26.358,-179.9801,0.0404,0.0000
C00591=-88.507,45.948,26.301,179.9207,-0.1105,0.0000
C00592=-86.297,48.509,26.245,-179.2986,0.6720,0.0000
C00593=-84.010,50.266,26.175,-177.6750,1.3092,0.0000
C00594=-81.959,51.029,26.043,-175.6775,0.9255,0.0000
C00595=-79.995,51.336,25.771,-171.8841,0.8549,0.0000
C00596=-78.105,51.679,25.406,-164.9814,3.3027,0.0000
C00597=-76.218,52.487,25.041,-158.0702,11.7507,0.0000
C00598=-74.059,54.287,24.767,-157.3747,22.2371,0.0000
C00599=-71.231,57.528,24.657,-158.2376,25.2298,0.0000
C00600=-68.184,61.085,24.652,-157.5713,24.8132,0.0000
C00601=-64.734,64.734,24.655,-156.3440,23.6556,0.0000
C00602=-61.085,68.184,24.652,-155.1871,22.4290,0.0000
C00603=-57.528,71.231,24.657,-154.7707,21.7628,0.0000
C00604=-54.287,74.059,24.767,-157.7626,22.6250,0.0000
C00605=-52.487,76.218,25.041,-168.2493,21.9298,0.0000
C00606=-51.679,78.105,25.406,-176.6973,15.0186,0.0000
C00607=-51.336,79.995,25.771,-179.1451,8.1159,0.0000
C00608=-51.029,81.959,26.043,-179.0745,4.3225,0.0000
C00609=-50.266,84.010,26.175,-178.6908,2.3250,0.0000
C00610=-48.509,86.297,26.245,-179.3280,0.7014,0.0000
C00611=-45.948,88.507,26.301,179.8895,-0.0793,0.0000
C00612=-42.931,90.273,26.358,-179.9596,0.0199,0.0000
C00613=-39.829,91.721,26.395,-179.9960,0.0018,0.0000
C00614=-36.693,93.020,26.395,-179.9960,0.0016,0.0000
C00615=-33.476,94.189,26.358,-179.9573,0.0145,0.0000
C00616=-30.093,95.074,26.301,179.8658,-0.0220,0.0000
C00617=-26.720,95.323,26.245,-179.0289,-0.0208,0.0000
C00618=-23.861,94.948,26.175,-177.4309,-0.7190,0.0000
C00619=-21.871,94.037,26.043,-176.2884,-2.4064,0.0000
C00620=-20.265,92.865,25.771,-173.6442,-5.1590,0.0000
C00621=-18.686,91.772,25.406,-167.0189,-8.4697,0.0000
C00622=-16.781,91.008,25.041,-156.6468,-7.8344,0.0000
C00623=-13.981,90.755,24.767,-149.7234,-0.3207,0.0000
C00624=-9.690,91.047,24.657,-148.3889,2.9133,0.0000
C00625=-5.020,91.408,24.652,-148.2512,2.0077,0.0000
C00626=0.000,91.548,24.655,-148.2220,0.0004,0.0000
C00627=0.000,90.369,26.513,-146.9909,0.0004,0.0000
C00628=4.912,90.233,26.509,-147.0206,-2.0967,0.0000
C00629=9.508,89.882,26.515,-147.1605,-2.8971,0.0000
C00630=13.759,89.629,26.645,-148.6809,1.2171,0.0000
C00631=16.509,89.983,26.968,-157.2655,9.5618,0.0000
C00632=18.373,90.901,27.402,-168.7365,8.8492,0.0000
C00633=19.923,92.196,27.838,-175.1312,4.7417,0.0000
C00634=21.502,93.597,28.166,-177.5251,1.9666,0.0000
C00635=23.458,94.728,28.327,-178.2716,0.6326,0.0000
C00636=26.340,95.277,28.411,-179.4215,0.0370,0.0000
C00637=29.791,95.129,28.479,179.6935,0.0440,0.0000
C00638=33.285,94.252,28.548,-179.9707,-0.0099,0.0000
C00639=36.628,93.045,28.594,-179.9976,-0.0009,0.0000
C00640=39.893,91.693,28.594,-179.9976,-0.0010,0.0000
C00641=43.110,90.182,28.548,-179.9723,-0.0138,0.0000
C00642=46.201,88.332,28.479,179.7522,0.1856,0.0000
C00643=48.746,85.996,28.411,-179.6171,-0.4352,0.0000
C00644=50.396,83.570,28.327,-179.2249,-1.6694,0.0000
C00645=50.979,81.387,28.166,-179.6401,-3.1392,0.0000
C00646=51.105,79.281,27.838,-179.9095,-6.7798,0.0000
C00647=51.285,77.269,27.402,-178.2394,-14.0854,0.0000
C00648=51.954,75.301,26.968,-169.9528,-22.5582,0.0000
C00649=53.649,73.106,26.645,-157.4504,-24.0022,0.0000
C00650=56.833,70.280,26.515,-153.7948,-22.8119,0.0000
C00651=60.331,67.277,26.509,-154.1393,-23.4102,0.0000
C00652=63.901,63.901,26.513,-155.3281,-24.6724,0.0000
C00653=67.277,60.331,26.509,-156.5894,-25.8604,0.0000
C00654=70.280,56.833,26.515,-157.1876,-26.2046,0.0000
C00655=73.106,53.649,26.645,-155.9981,-22.5500,0.0000
C00656=75.301,51.954,26.968,-157.4418,-10.0472,0.0000
C00657=77.269,51.285,27.402,-165.9146,-1.7606,0.0000
C00658=79.281,51.105,27.838,-173.2202,-0.0905,0.0000
C00659=81.387,50.979,28.166,-176.8608,-0.3599,0.0000
C00660=83.570,50.396,28.327,-178.3306,-0.7751,0.0000
C00661=85.996,48.746,28.411,-179.5648,-0.3829,0.0000
C00662=88.332,46.201,28.479,179.8144,0.2478,0.0000
C00663=90.182,43.110,28.548,-179.9862,-0.0277,0.0000
C00664=91.693,39.893,28.594,-179.9990,-0.0024,0.0000
C00665=93.045,36.628,28.594,-179.9991,-0.0024,0.0000
C00666=94.252,33.285,28.548,-179.9901,-0.0293,0.0000
C00667=95.129,29.791,28.479,179.9560,0.3065,0.0000
C00668=95.277,26.340,28.411,179.9630,-0.5785,0.0000
C00669=94.728,23.458,28.327,179.3674,-1.7284,0.0000
C00670=93.597,21.502,28.166,178.0334,-2.4749,0.0000
C00671=92.196,19.923,27.838,175.2583,-4.8688,0.0000
C00672=90.901,18.373,27.402,171.1508,-11.2635,0.0000
C00673=89.983,16.509,26.968,170.4382,-22.7345,0.0000
C00674=89.629,13.759,26.645,178.7829,-31.3191,0.0000
C00675=89.882,9.508,26.515,-177.1029,-32.8395,0.0000
C00676=90.233,4.912,26.509,-177.9033,-32.9794,0.0000
C00677=90.369,0.000,26.513,179.9996,-33.0091,0.0000
C00678=90.233,-4.912,26.509,177.9038,-32.9794,0.0000
C00679=89.882,-9.508,26.515,177.1039,-32.8395,0.0000
C00680=89.629,-13.759,26.645,-178.7835,-31.3192,0.0000
C00681=89.983,-16.509,26.968,-170.4382,-22.7345,0.0000
C00682=90.901,-18.373,27.402,-171.1508,-11.2635,0.0000
C00683=92.196,-19.923,27.838,-175.2583,-4.8688,0.0000
C00684=93.597,-21.502,28.166,-178.0334,-2.4749,0.0000
C00685=94.728,-23.458,28.327,-179.3674,-1.7284,0.0000
C00686=95.277,-26.340,28.411,-179.9630,-0.5785,0.0000
C00687=95.129,-29.791,28.479,-179.9560,0.3065,0.0000
C00688=94.252,-33.285,28.548,179.9901,-0.0293,0.0000
C00689=93.045,-36.628,28.594,179.9991,-0.0024,0.0000
C00690=91.693,-39.893,28.594,179.9990,-0.0024,0.0000
C00691=90.182,-43.110,28.548,179.9862,-0.0277,0.0000
C00692=88.332,-46.201,28.479,-179.8144,0.2478,0.0000
C00693=85.996,-48.746,28.411,179.5648,-0.3829,0.0000
C00694=83.570,-50.396,28.327,178.3306,-0.7751,0.0000
C00695=81.387,-50.979,28.166,176.8608,-0.3599,0.0000
C00696=79.281,-51.105,27.838,173.2202,-0.0905,0.0000
C00697=77.269,-51.285,27.402,165.9146,-1.7606,0.0000
C00698=75.301,-51.954,26.968,157.4418,-10.0472,0.0000
C00699=73.106,-53.649,26.645,155.9978,-22.5496,0.0000
C00700=70.280,-56.833,26.515,157.1881,-26.2052,0.0000
C00701=67.277,-60.331,26.509,156.5898,-25.8607,0.0000
C00702=63.901,-63.901,26.513,155.3276,-24.6719,0.0000
C00703=60.331,-67.277,26.509,154.1396,-23.4106,0.0000
C00704=56.833,-70.280,26.515,153.7954,-22.8124,0.0000
C00705=53.649,-73.106,26.645,157.4500,-24.0019,0.0000
C00706=51.954,-75.301,26.968,169.9528,-22.5582,0.0000
C00707=51.285,-77.269,27.402,178.2394,-14.0854,0.0000
C00708=51.105,-79.281,27.838,179.9095,-6.7798,0.0000
C00709=50.979,-81.387,28.166,179.6401,-3.1392,0.0000
C00710=50.396,-83.570,28.327,179.2249,-1.6694,0.0000
C00711=48.746,-85.996,28.411,179.6171,-0.4352,0.0000
C00712=46.201,-88.332,28.479,-179.7522,0.1856,0.0000
C00713=43.110,-90.182,28.548,179.9723,-0.0138,0.0000
C00714=39.893,-91.693,28.594,179.9976,-0.0010,0.0000
C00715=36.628,-93.045,28.594,179.9976,-0.0009,0.0000
C00716=33.285,-94.252,28.548,179.9707,-0.0099,0.0000
C00717=29.791,-95.129,28.479,-179.6935,0.0440,0.0000
C00718=26.340,-95.277,28.411,179.4215,0.0370,0.0000
C00719=23.458,-94.728,28.327,178.2716,0.6326,0.0000
C00720=21.502,-93.597,28.166,177.5251,1.9666,0.0000
C00721=19.923,-92.196,27.838,175.1312,4.7417,0.0000
C00722=18.373,-90.901,27.402,168.7365,8.8492,0.0000
C00723=16.509,-89.983,26.968,157.2655,9.5618,0.0000
C00724=13.759,-89.629,26.645,148.6809,1.2171,0.0000
C00725=9.508,-89.882,26.515,147.1605,-2.8971,0.0000
C00726=4.912,-90.233,26.509,147.0206,-2.0967,0.0000
C00727=0.000,-90.369,26.513,146.9909,0.0004,0.0000
C00728=0.000,-90.369,26.513,146.9909,0.0004,0.0000
C00729=-4.912,-90.233,26.509,147.0206,2.0962,0.0000
C00730=-9.508,-89.882,26.515,147.1605,2.8961,0.0000
C00731=-13.759,-89.629,26.645,148.6808,-1.2165,0.0000
C00732=-16.509,-89.983,26.968,157.2655,-9.5618,0.0000
C00733=-18.373,-90.901,27.402,168.7365,-8.8492,0.0000
C00734=-19.923,-92.196,27.838,175.1312,-4.7417,0.0000
C00735=-21.502,-93.597,28.166,177.5251,-1.9666,0.0000
C00736=-23.458,-94.728,28.327,178.2716,-0.6326,0.0000
C00737=-26.340,-95.277,28.411,179.4215,-0.0370,0.0000
C00738=-29.791,-95.129,28.479,-179.6935,-0.0440,0.0000
C00739=-33.285,-94.252,28.548,179.9707,0.0099,0.0000
C00740=-36.628,-93.045,28.594,179.9976,0.0009,0.0000
C00741=-39.893,-91.693,28.594,179.9976,0.0010,0.0000
C00742=-43.110,-90.182,28.548,179.9723,0.0138,0.0000
C00743=-46.201,-88.332,28.479,-179.7522,-0.1856,0.0000
C00744=-48.746,-85.996,28.411,179.6171,0.4352,0.0000
C00745=-50.396,-83.570,28.327,179.2249,1.6694,0.0000
C00746=-50.979,-81.387,28.166,179.6401,3.1392,0.0000
C00747=-51.105,-79.281,27.838,179.9095,6.7798,0.0000
C00748=-51.285,-77.269,27.402,178.2394,14.0854,0.0000
C00749=-51.954,-75.301,26.968,169.9528,22.5582,0.0000
C00750=-53.649,-73.106,26.645,157.4504,24.0022,0.0000
C00751=-56.833,-70.280,26.515,153.7948,22.8119,0.0000
C00752=-60.331,-67.277,26.509,154.1393,23.4102,0.0000
C00753=-63.901,-63.901,26.513,155.3281,24.6724,0.0000
C00754=-67.277,-60.331,26.509,156.5894,25.8604,0.0000
C00755=-70.280,-56.833,26.515,157.1876,26.2046,0.0000
C00756=-73.106,-53.649,26.645,155.9981,22.5500,0.0000
C00757=-75.301,-51.954,26.968,157.4418,10.0472,0.0000
C00758=-77.269,-51.285,27.402,165.9146,1.7606,0.0000
C00759=-79.281,-51.105,27.838,173.2202,0.0905,0.0000
C00760=-81.387,-50.979,28.166,176.8608,0.3599,0.0000
C00761=-83.570,-50.396,28.327,178.3306,0.7751,0.0000
C00762=-85.996,-48.746,28.411,179.5648,0.3829,0.0000
C00763=-88.332,-46.201,28.479,-179.8144,-0.2478,0.0000
C00764=-90.182,-43.110,28.548,179.9862,0.0277,0.0000
C00765=-91.693,-39.893,28.594,179.9990,0.0024,0.0000
C00766=-93.045,-36.628,28.594,179.9991,0.0024,0.0000
C00767=-94.252,-33.285,28.548,179.9901,0.0293,0.0000
C00768=-95.129,-29.791,28.479,-179.9560,-0.3065,0.0000
C00769=-95.277,-26.340,28.411,-179.9630,0.5785,0.0000
C00770=-94.728,-23.458,28.327,-179.3674,1.7284,0.0000
C00771=-93.597,-21.502,28.166,-178.0334,2.4749,0.0000
C00772=-92.196,-19.923,27.838,-175.2583,4.8688,0.0000
C00773=-90.901,-18.373,27.402,-171.1508,11.2635,0.0000
C00774=-89.983,-16.509,26.968,-170.4382,22.7345,0.0000
C00775=-89.629,-13.759,26.645,-178.7829,31.3191,0.0000
C00776=-89.882,-9.508,26.515,177.1029,32.8395,0.0000
C00777=-90.233,-4.912,26.509,177.9033,32.9794,0.0000
C00778=-90.369,0.000,26.513,-179.9996,33.0091,0.0000
C00779=-90.233,4.912,26.509,-177.9038,32.9794,0.0000
C00780=-89.882,9.508,26.515,-177.1039,32.8395,0.0000
C00781=-89.629,13.759,26.645,178.7835,31.3192,0.0000
C00782=-89.983,16.509,26.968,170.4382,22.7345,0.0000
C00783=-90.901,18.373,27.402,171.1508,11.2635,0.0000
C00784=-92.196,19.923,27.838,175.2583,4.8688,0.0000
C00785=-93.597,21.502,28.166,178.0334,2.4749,0.0000
C00786=-94.728,23.458,28.327,179.3674,1.7284,0.0000
C00787=-95.277,26.340,28.411,179.9630,0.5785,0.0000
C00788=-95.129,29.791,28.479,179.9560,-0.3065,0.0000
C00789=-94.252,33.285,28.548,-179.9901,0.0293,0.0000
C00790=-93.045,36.628,28.594,-179.9991,0.0024,0.0000
C00791=-91.693,39.893,28.594,-179.9990,0.0024,0.0000
C00792=-90.182,43.110,28.548,-179.9862,0.0277,0.0000
C00793=-88.332,46.201,28.479,179.8144,-0.2478,0.0000
C00794=-85.996,48.746,28.411,-179.5648,0.3829,0.0000
C00795=-83.570,50.396,28.327,-178.3306,0.7751,0.0000
C00796=-81.387,50.979,28.166,-176.8608,0.3599,0.0000
C00797=-79.281,51.105,27.838,-173.2202,0.0905,0.0000
C00798=-77.269,51.285,27.402,-165.9146,1.7606,0.0000
C00799=-75.301,51.954,26.968,-157.4418,10.0472,0.0000
C00800=-73.106,53.649,26.645,-155.9978,22.5496,0.0000
C00801=-70.280,56.833,26.515,-157.1881,26.2052,0.0000
C00802=-67.277,60.331,26.509,-156.5898,25.8607,0.0000
C00803=-63.901,63.901,26.513,-155.3276,24.6719,0.0000
C00804=-60.331,67.277,26.509,-154.1396,23.4106,0.0000
C00805=-56.833,70.280,26.515,-153.7954,22.8124,0.0000
C00806=-53.649,73.106,26.645,-157.4500,24.0019,0.0000
C00807=-51.954,75.301,26.968,-169.9528,22.5582,0.0000
C00808=-51.285,77.269,27.402,-178.2394,14.0854,0.0000
C00809=-51.105,79.281,27.838,-179.9095,6.7798,0.0000
C00810=-50.979,81.387,28.166,-179.6401,3.1392,0.0000
C00811=-50.396,83.570,28.327,-179.2249,1.6694,0.0000
C00812=-48.746,85.996,28.411,-179.6171,0.4352,0.0000
C00813=-46.201,88.332,28.479,179.7522,-0.1856,0.0000
C00814=-43.110,90.182,28.548,-179.9723,0.0138,0.0000
C00815=-39.893,91.693,28.594,-179.9976,0.0010,0.0000
C00816=-36.628,93.045,28.594,-179.9976,0.0009,0.0000
C00817=-33.285,94.252,28.548,-179.9707,0.0099,0.0000
C00818=-29.791,95.129,28.479,179.6935,-0.0440,0.0000
C00819=-26.340,95.277,28.411,-179.4215,-0.0370,0.0000
C00820=-23.458,94.728,28.327,-178.2716,-0.6326,0.0000
C00821=-21.502,93.597,28.166,-177.5251,-1.9666,0.0000
C00822=-19.923,92.196,27.838,-175.1312,-4.7417,0.0000
C00823=-18.373,90.901,27.402,-168.7365,-8.8492,0.0000
C00824=-16.509,89.983,26.968,-157.2655,-9.5618,0.0000
C00825=-13.759,89.629,26.645,-148.6808,-1.2165,0.0000
C00826=-9.508,89.882,26.515,-147.1605,2.8961,0.0000
C00827=-4.912,90.233,26.509,-147.0206,2.0962,0.0000
C00828=0.000,90.369,26.513,-146.9909,0.0004,0.0000
C00829=0.000,89.153,28.346,-145.9022,0.0004,0.0000
C00830=4.801,89.020,28.341,-145.9323,-2.1748,0.0000
C00831=9.321,88.681,28.348,-146.0749,-2.8439,0.0000
C00832=13.530,88.468,28.499,-147.8255,2.2168,0.0000
C00833=16.227,88.922,28.874,-158.3138,11.0586,0.0000
C00834=18.049,89.999,29.382,-170.5154,8.7916,0.0000
C00835=19.567,91.502,29.895,-176.4765,4.0373,0.0000
C00836=21.117,93.139,30.283,-178.6645,1.2702,0.0000
C00837=23.038,94.499,30.474,-179.1703,0.3790,0.0000
C00838=25.943,95.229,30.574,-179.8563,0.0154,0.0000
C00839=29.476,95.186,30.656,179.5089,0.0604,0.0000
C00840=33.085,94.318,30.738,-179.9851,-0.0050,0.0000
C00841=36.560,93.071,30.793,-179.9993,-0.0003,0.0000
C00842=39.959,91.663,30.793,-179.9994,-0.0003,0.0000
C00843=43.298,90.088,30.738,-179.9860,-0.0070,0.0000
C00844=46.464,88.150,30.656,179.6100,0.3045,0.0000
C00845=48.993,85.682,30.574,-179.9092,-0.1125,0.0000
C00846=50.531,83.111,30.474,-179.6813,-0.8547,0.0000
C00847=50.927,80.791,30.283,-179.9538,-1.8423,0.0000
C00848=50.865,78.538,29.895,179.6351,-5.3387,0.0000
C00849=50.876,76.401,29.382,-179.4973,-12.8163,0.0000
C00850=51.403,74.351,28.874,-171.8620,-22.7528,0.0000
C00851=52.989,72.123,28.499,-157.3406,-25.2777,0.0000
C00852=56.115,69.298,28.348,-152.9451,-23.7726,0.0000
C00853=59.552,66.342,28.341,-153.2053,-24.2903,0.0000
C00854=63.040,63.040,28.346,-154.4195,-25.5810,0.0000
C00855=66.342,59.552,28.341,-155.7093,-26.7944,0.0000
C00856=69.298,56.115,28.348,-156.2269,-27.0542,0.0000
C00857=72.123,52.989,28.499,-154.7226,-22.6600,0.0000
C00858=74.351,51.403,28.874,-157.2472,-8.1380,0.0000
C00859=76.401,50.876,29.382,-167.1837,-0.5027,0.0000
C00860=78.538,50.865,29.895,-174.6613,0.3649,0.0000
C00861=80.791,50.927,30.283,-178.1577,-0.0462,0.0000
C00862=83.111,50.531,30.474,-179.1453,-0.3187,0.0000
C00863=85.682,48.993,30.574,-179.8875,-0.0908,0.0000
C00864=88.150,46.464,30.656,179.6955,0.3900,0.0000
C00865=90.088,43.298,30.738,-179.9930,-0.0140,0.0000
C00866=91.663,39.959,30.793,-179.9997,-0.0006,0.0000
C00867=93.071,36.560,30.793,-179.9997,-0.0007,0.0000
C00868=94.318,33.085,30.738,-179.9950,-0.0149,0.0000
C00869=95.186,29.476,30.656,179.9396,0.4911,0.0000
C00870=95.229,25.943,30.574,179.9846,-0.1437,0.0000
C00871=94.499,23.038,30.474,179.6210,-0.8297,0.0000
C00872=93.139,21.117,30.283,178.7298,-1.3355,0.0000
C00873=91.502,19.567,29.895,175.9627,-3.5235,0.0000
C00874=89.999,18.049,29.382,171.2084,-9.4846,0.0000
C00875=88.922,16.227,28.874,168.9414,-21.6862,0.0000
C00876=88.468,13.530,28.499,177.7832,-32.1745,0.0000
C00877=88.681,9.321,28.348,-177.1561,-33.9251,0.0000
C00878=89.020,4.801,28.341,-177.8252,-34.0677,0.0000
C00879=89.153,0.000,28.346,179.9996,-34.0978,0.0000
C00880=89.020,-4.801,28.341,177.8258,-34.0678,0.0000
C00881=88.681,-9.321,28.348,177.1572,-33.9251,0.0000
C00882=88.468,-13.530,28.499,-177.7839,-32.1746,0.0000
C00883=88.922,-16.227,28.874,-168.9414,-21.6862,0.0000
C00884=89.999,-18.049,29.382,-171.2084,-9.4846,0.0000
C00885=91.502,-19.567,29.895,-175.9627,-3.5235,0.0000
C00886=93.139,-21.117,30.283,-178.7298,-1.3355,0.0000
C00887=94.499,-23.038,30.474,-179.6210,-0.8297,0.0000
C00888=95.229,-25.943,30.574,-179.9846,-0.1437,0.0000
C00889=95.186,-29.476,30.656,-179.9396,0.4911,0.0000
C00890=94.318,-33.085,30.738,179.9950,-0.0149,0.0000
C00891=93.071,-36.560,30.793,179.9997,-0.0007,0.0000
C00892=91.663,-39.959,30.793,179.9997,-0.0006,0.0000
C00893=90.088,-43.298,30.738,179.9930,-0.0140,0.0000
C00894=88.150,-46.464,30.656,-179.6955,0.3900,0.0000
C00895=85.682,-48.993,30.574,179.8875,-0.0908,0.0000
C00896=83.111,-50.531,30.474,179.1453,-0.3187,0.0000
C00897=80.791,-50.927,30.283,178.1577,-0.0462,0.0000
C00898=78.538,-50.865,29.895,174.6613,0.3649,0.0000
C00899=76.401,-50.876,29.382,167.1837,-0.5027,0.0000
C00900=74.351,-51.403,28.874,157.2472,-8.1380,0.0000
C00901=72.123,-52.989,28.499,154.7223,-22.6594,0.0000
C00902=69.298,-56.115,28.348,156.2274,-27.0549,0.0000
C00903=66.342,-59.552,28.341,155.7097,-26.7947,0.0000
C00904=63.040,-63.040,28.346,154.4190,-25.5805,0.0000
C00905=59.552,-66.342,28.341,153.2056,-24.2907,0.0000
C00906=56.115,-69.298,28.348,152.9458,-23.7731,0.0000
C00907=52.989,-72.123,28.499,157.3400,-25.2774,0.0000
C00908=51.403,-74.351,28.874,171.8620,-22.7528,0.0000
C00909=50.876,-76.401,29.382,179.4973,-12.8163,0.0000
C00910=50.865,-78.538,29.895,-179.6351,-5.3387,0.0000
C00911=50.927,-80.791,30.283,179.9538,-1.8423,0.0000
C00912=50.531,-83.111,30.474,179.6813,-0.8547,0.0000
C00913=48.993,-85.682,30.574,179.9092,-0.1125,0.0000
C00914=46.464,-88.150,30.656,-179.6100,0.3045,0.0000
C00915=43.298,-90.088,30.738,179.9860,-0.0070,0.0000
C00916=39.959,-91.663,30.793,179.9994,-0.0003,0.0000
C00917=36.560,-93.071,30.793,179.9993,-0.0003,0.0000
C00918=33.085,-94.318,30.738,179.9851,-0.0050,0.0000
C00919=29.476,-95.186,30.656,-179.5089,0.0604,0.0000
C00920=25.943,-95.229,30.574,179.8563,0.0154,0.0000
C00921=23.038,-94.499,30.474,179.1703,0.3790,0.0000
C00922=21.117,-93.139,30.283,178.6645,1.2702,0.0000
C00923=19.567,-91.502,29.895,176.4765,4.0373,0.0000
C00924=18.049,-89.999,29.382,170.5154,8.7916,0.0000
C00925=16.227,-88.922,28.874,158.3138,11.0586,0.0000
C00926=13.530,-88.468,28.499,147.8255,2.2168,0.0000
C00927=9.321,-88.681,28.348,146.0749,-2.8439,0.0000
C00928=4.801,-89.020,28.341,145.9323,-2.1748,0.0000
C00929=0.000,-89.153,28.346,145.9022,0.0004,0.0000
C00930=0.000,-89.153,28.346,145.9022,0.0004,0.0000
C00931=-4.801,-89.020,28.341,145.9322,2.1742,0.0000
C00932=-9.321,-88.681,28.348,146.0749,2.8428,0.0000
C00933=-13.530,-88.468,28.499,147.8254,-2.2161,0.0000
C00934=-16.227,-88.922,28.874,158.3138,-11.0586,0.0000
C00935=-18.049,-89.999,29.382,170.5154,-8.7916,0.0000
C00936=-19.567,-91.502,29.895,176.4765,-4.0373,0.0000
C00937=-21.117,-93.139,30.283,178.6645,-1.2702,0.0000
C00938=-23.038,-94.499,30.474,179.1703,-0.3790,0.0000
C00939=-25.943,-95.229,30.574,179.8563,-0.0154,0.0000
C00940=-29.476,-95.186,30.656,-179.5089,-0.0604,0.0000
C00941=-33.085,-94.318,30.738,179.9851,0.0050,0.0000
C00942=-36.560,-93.071,30.793,179.9993,0.0003,0.0000
C00943=-39.959,-91.663,30.793,179.9994,0.0003,0.0000
C00944=-43.298,-90.088,30.738,179.9860,0.0070,0.0000
C00945=-46.464,-88.150,30.656,-179.6100,-0.3045,0.0000
C00946=-48.993,-85.682,30.574,179.9092,0.1125,0.0000
C00947=-50.531,-83.111,30.474,179.6813,0.8547,0.0000
C00948=-50.927,-80.791,30.283,179.9538,1.8423,0.0000
C00949=-50.865,-78.538,29.895,-179.6351,5.3387,0.0000
C00950=-50.876,-76.401,29.382,179.4973,12.8163,0.0000
C00951=-51.403,-74.351,28.874,171.8620,22.7528,0.0000
C00952=-52.989,-72.123,28.499,157.3406,25.2777,0.0000
C00953=-56.115,-69.298,28.348,152.9451,23.7726,0.0000
C00954=-59.552,-66.342,28.341,153.2053,24.2903,0.0000
C00955=-63.040,-63.040,28.346,154.4195,25.5810,0.0000
C00956=-66.342,-59.552,28.341,155.7093,26.7944,0.0000
C00957=-69.298,-56.115,28.348,156.2269,27.0542,0.0000
C00958=-72.123,-52.989,28.499,154.7226,22.6600,0.0000
C00959=-74.351,-51.403,28.874,157.2472,8.1380,0.0000
C00960=-76.401,-50.876,29.382,167.1837,0.5027,0.0000
C00961=-78.538,-50.865,29.895,174.6613,-0.3649,0.0000
C00962=-80.791,-50.927,30.283,178.1577,0.0462,0.0000
C00963=-83.111,-50.531,30.474,179.1453,0.3187,0.0000
C00964=-85.682,-48.993,30.574,179.8875,0.0908,0.0000
C00965=-88.150,-46.464,30.656,-179.6955,-0.3900,0.0000
C00966=-90.088,-43.298,30.738,179.9930,0.0140,0.0000
C00967=-91.663,-39.959,30.793,179.9997,0.0006,0.0000
C00968=-93.071,-36.560,30.793,179.9997,0.0007,0.0000
C00969=-94.318,-33.085,30.738,179.9950,0.0149,0.0000
C00970=-95.186,-29.476,30.656,-179.9396,-0.4911,0.0000
C00971=-95.229,-25.943,30.574,-179.9846,0.1437,0.0000
C00972=-94.499,-23.038,30.474,-179.6210,0.8297,0.0000
C00973=-93.139,-21.117,30.283,-178.7298,1.3355,0.0000
C00974=-91.502,-19.567,29.895,-175.9627,3.5235,0.0000
C00975=-89.999,-18.049,29.382,-171.2084,9.4846,0.0000
C00976=-88.922,-16.227,28.874,-168.9414,21.6862,0.0000
C00977=-88.468,-13.530,28.499,-177.7832,32.1745,0.0000
C00978=-88.681,-9.321,28.348,177.1561,33.9251,0.0000
C00979=-89.020,-4.801,28.341,177.8252,34.0677,0.0000
C00980=-89.153,0.000,28.346,-179.9996,34.0978,0.0000
C00981=-89.020,4.801,28.341,-177.8258,34.0678,0.0000
C00982=-88.681,9.321,28.348,-177.1572,33.9251,0.0000
C00983=-88.468,13.530,28.499,177.7839,32.1746,0.0000
C00984=-88.922,16.227,28.874,168.9414,21.6862,0.0000
C00985=-89.999,18.049,29.382,171.2084,9.4846,0.0000
C00986=-91.502,19.567,29.895,175.9627,3.5235,0.0000
C00987=-93.139,21.117,30.283,178.7298,1.3355,0.0000
C00988=-94.499,23.038,30.474,179.6210,0.8297,0.0000
C00989=-95.229,25.943,30.574,179.9846,0.1437,0.0000
C00990=-95.186,29.476,30.656,179.9396,-0.4911,0.0000
C00991=-94.318,33.085,30.738,-179.9950,0.0149,0.0000
C00992=-93.071,36.560,30.793,-179.9997,0.0007,0.0000
C00993=-91.663,39.959,30.793,-179.9997,0.0006,0.0000
C00994=-90.088,43.298,30.738,-179.9930,0.0140,0.0000
C00995=-88.150,46.464,30.656,179.6955,-0.3900,0.0000
C00996=-85.682,48.993,30.574,-179.8875,0.0908,0.0000
C00997=-83.111,50.531,30.474,-179.1453,0.3187,0.0000
C00998=-80.791,50.927,30.283,-178.1577,0.0462,0.0000
C00999=-78.538,50.865,29.895,-174.6613,-0.3649,0.0000
C01000=-76.401,50.876,29.382,-167.1837,0.5027,0.0000
C01001=-74.351,51.403,28.874,-157.2472,8.1380,0.0000
C01002=-72.123,52.989,28.499,-154.7223,22.6594,0.0000
C01003=-69.298,56.115,28.348,-156.2274,27.0549,0.0000
C01004=-66.342,59.552,28.341,-155.7097,26.7947,0.0000
C01005=-63.040,63.040,28.346,-154.4190,25.5805,0.0000
C01006=-59.552,66.342,28.341,-153.2056,24.2907,0.0000
C01007=-56.115,69.298,28.348,-152.9458,23.7731,0.0000
C01008=-52.989,72.123,28.499,-157.3400,25.2774,0.0000
C01009=-51.403,74.351,28.874,-171.8620,22.7528,0.0000
C01010=-50.876,76.401,29.382,-179.4973,12.8163,0.0000
C01011=-50.865,78.538,29.895,179.6351,5.3387,0.0000
C01012=-50.927,80.791,30.283,-179.9538,1.8423,0.0000
C01013=-50.531,83.111,30.474,-179.6813,0.8547,0.0000
C01014=-48.993,85.682,30.574,-179.9092,0.1125,0.0000
C01015=-46.464,88.150,30.656,179.6100,-0.3045,0.0000
C01016=-43.298,90.088,30.738,-179.9860,0.0070,0.0000
C01017=-39.959,91.663,30.793,-179.9994,0.0003,0.0000
C01018=-36.560,93.071,30.793,-179.9993,0.0003,0.0000
C01019=-33.085,94.318,30.738,-179.9851,0.0050,0.0000
C01020=-29.476,95.186,30.656,179.5089,-0.0604,0.0000
C01021=-25.943,95.229,30.574,-179.8563,-0.0154,0.0000
C01022=-23.038,94.499,30.474,-179.1703,-0.3790,0.0000
C01023=-21.117,93.139,30.283,-178.6645,-1.2702,0.0000
C01024=-19.567,91.502,29.895,-176.4765,-4.0373,0.0000
C01025=-18.049,89.999,29.382,-170.5154,-8.7916,0.0000
C01026=-16.227,88.922,28.874,-158.3138,-11.0586,0.0000
C01027=-13.530,88.468,28.499,-147.8254,-2.2161,0.0000
C01028=-9.321,88.681,28.348,-146.0749,2.8428,0.0000
C01029=-4.801,89.020,28.341,-145.9322,2.1742,0.0000
C01030=0.000,89.153,28.346,-145.9022,0.0004,0.0000
C01031=0.000,87.904,30.157,-144.9432,0.0004,0.0000
C01032=4.687,87.776,30.152,-144.9734,-2.2427,0.0000
C01033=9.129,87.447,30.160,-145.1196,-2.7561,0.0000
C01034=13.294,87.274,30.332,-147.1504,3.3033,0.0000
C01035=15.938,87.830,30.762,-159.7282,12.2356,0.0000
C01036=17.714,89.068,31.347,-172.2272,8.3691,0.0000
C01037=19.200,90.783,31.942,-177.6276,3.1482,0.0000
C01038=20.718,92.664,32.394,-179.6431,0.3988,0.0000
C01039=22.602,94.262,32.617,179.9322,-0.0374,0.0000
C01040=25.531,95.180,32.735,179.6818,-0.0477,0.0000
C01041=29.149,95.246,32.831,179.3160,0.0705,0.0000
C01042=32.878,94.386,32.928,179.9997,0.0001,0.0000
C01043=36.490,93.098,32.991,179.9988,0.0004,0.0000
C01044=40.028,91.633,32.991,179.9989,0.0005,0.0000
C01045=43.493,89.989,32.928,179.9997,0.0001,0.0000
C01046=46.737,87.960,32.831,179.4665,0.4338,0.0000
C01047=49.249,85.356,32.735,179.8087,0.2587,0.0000
C01048=50.671,82.635,32.617,179.9785,0.0744,0.0000
C01049=50.874,80.174,32.394,179.9703,-0.5344,0.0000
C01050=50.617,77.770,31.942,179.4502,-3.9008,0.0000
C01051=50.455,75.506,31.347,179.5699,-11.3401,0.0000
C01052=50.836,73.375,30.762,-173.8456,-22.5147,0.0000
C01053=52.312,71.113,30.332,-157.4247,-26.4448,0.0000
C01054=55.379,68.290,30.160,-152.2123,-24.6497,0.0000
C01055=58.753,65.381,30.152,-152.3768,-25.0757,0.0000
C01056=62.157,62.157,30.157,-153.6112,-26.3893,0.0000
C01057=65.381,58.753,30.152,-154.9239,-27.6229,0.0000
C01058=68.290,55.379,30.160,-155.3497,-27.7869,0.0000
C01059=71.113,52.312,30.332,-153.5556,-22.5759,0.0000
C01060=73.375,50.836,30.762,-157.4853,-6.1544,0.0000
C01061=75.506,50.455,31.347,-168.6599,0.4301,0.0000
C01062=77.770,50.617,31.942,-176.0992,0.5498,0.0000
C01063=80.174,50.874,32.394,-179.4656,0.0297,0.0000
C01064=82.635,50.671,32.617,179.9256,0.0215,0.0000
C01065=85.356,49.249,32.735,179.7413,0.1913,0.0000
C01066=87.960,46.737,32.831,179.5662,0.5335,0.0000
C01067=89.989,43.493,32.928,179.9999,0.0003,0.0000
C01068=91.633,40.028,32.991,179.9995,0.0011,0.0000
C01069=93.098,36.490,32.991,179.9996,0.0012,0.0000
C01070=94.386,32.878,32.928,179.9999,0.0003,0.0000
C01071=95.246,29.149,32.831,179.9295,0.6840,0.0000
C01072=95.180,25.531,32.735,-179.9523,0.3182,0.0000
C01073=94.262,22.602,32.617,-179.9626,0.0678,0.0000
C01074=92.664,20.718,32.394,179.6012,-0.3569,0.0000
C01075=90.783,19.200,31.942,176.8518,-2.3724,0.0000
C01076=89.068,17.714,31.347,171.6309,-7.7728,0.0000
C01077=87.830,15.938,30.762,167.7644,-20.2718,0.0000
C01078=87.274,13.294,30.332,176.6967,-32.8496,0.0000
C01079=87.447,9.129,30.160,-177.2439,-34.8804,0.0000
C01080=87.776,4.687,30.152,-177.7573,-35.0266,0.0000
C01081=87.904,0.000,30.157,179.9996,-35.0568,0.0000
C01082=87.776,-4.687,30.152,177.7578,-35.0266,0.0000
C01083=87.447,-9.130,30.160,177.2451,-34.8803,0.0000
C01084=87.274,-13.294,30.332,-176.6975,-32.8497,0.0000
C01085=87.830,-15.938,30.762,-167.7644,-20.2718,0.0000
C01086=89.068,-17.714,31.347,-171.6309,-7.7728,0.0000
C01087=90.783,-19.200,31.942,-176.8518,-2.3724,0.0000
C01088=92.664,-20.718,32.394,-179.6012,-0.3569,0.0000
C01089=94.262,-22.602,32.617,179.9626,0.0678,0.0000
C01090=95.180,-25.531,32.735,179.9523,0.3182,0.0000
C01091=95.246,-29.149,32.831,-179.9295,0.6840,0.0000
C01092=94.386,-32.878,32.928,-179.9999,0.0003,0.0000
C01093=93.098,-36.490,32.991,-179.9996,0.0012,0.0000
C01094=91.633,-40.028,32.991,-179.9995,0.0011,0.0000
C01095=89.989,-43.493,32.928,-179.9999,0.0003,0.0000
C01096=87.960,-46.737,32.831,-179.5662,0.5335,0.0000
C01097=85.356,-49.249,32.735,-179.7413,0.1913,0.0000
C01098=82.635,-50.671,32.617,-179.9256,0.0215,0.0000
C01099=80.174,-50.874,32.394,179.4656,0.0297,0.0000
C01100=77.770,-50.617,31.942,176.0992,0.5498,0.0000
C01101=75.506,-50.455,31.347,168.6599,0.4301,0.0000
C01102=73.375,-50.836,30.762,157.4853,-6.1544,0.0000
C01103=71.113,-52.312,30.332,153.5552,-22.5753,0.0000
C01104=68.290,-55.379,30.160,155.3503,-27.7877,0.0000
C01105=65.381,-58.753,30.152,154.9243,-27.6232,0.0000
C01106=62.157,-62.157,30.157,153.6107,-26.3888,0.0000
C01107=58.753,-65.381,30.152,152.3771,-25.0761,0.0000
C01108=55.379,-68.290,30.160,152.2131,-24.6503,0.0000
C01109=52.312,-71.113,30.332,157.4241,-26.4444,0.0000
C01110=50.836,-73.375,30.762,173.8456,-22.5147,0.0000
C01111=50.455,-75.506,31.347,-179.5699,-11.3401,0.0000
C01112=50.617,-77.770,31.942,-179.4502,-3.9008,0.0000
C01113=50.874,-80.174,32.394,-179.9703,-0.5344,0.0000
C01114=50.671,-82.635,32.617,-179.9785,0.0744,0.0000
C01115=49.249,-85.356,32.735,-179.8087,0.2587,0.0000
C01116=46.737,-87.960,32.831,-179.4665,0.4338,0.0000
C01117=43.493,-89.989,32.928,-179.9997,0.0001,0.0000
C01118=40.028,-91.633,32.991,-179.9989,0.0005,0.0000
C01119=36.490,-93.098,32.991,-179.9988,0.0004,0.0000
C01120=32.878,-94.386,32.928,-179.9997,0.0001,0.0000
C01121=29.149,-95.246,32.831,-179.3160,0.0705,0.0000
C01122=25.531,-95.180,32.735,-179.6818,-0.0477,0.0000
C01123=22.602,-94.262,32.617,-179.9322,-0.0374,0.0000
C01124=20.718,-92.664,32.394,179.6431,0.3988,0.0000
C01125=19.200,-90.783,31.942,177.6276,3.1482,0.0000
C01126=17.714,-89.068,31.347,172.2272,8.3691,0.0000
C01127=15.938,-87.830,30.762,159.7282,12.2356,0.0000
C01128=13.294,-87.274,30.332,147.1504,3.3033,0.0000
C01129=9.129,-87.447,30.160,145.1196,-2.7561,0.0000
C01130=4.687,-87.776,30.152,144.9734,-2.2427,0.0000
C01131=0.000,-87.904,30.157,144.9432,0.0004,0.0000
C01132=0.000,-87.904,30.157,144.9432,0.0004,0.0000
C01133=-4.687,-87.776,30.152,144.9734,2.2422,0.0000
C01134=-9.130,-87.447,30.160,145.1197,2.7549,0.0000
C01135=-13.294,-87.274,30.332,147.1503,-3.3025,0.0000
C01136=-15.938,-87.830,30.762,159.7282,-12.2356,0.0000
C01137=-17.714,-89.068,31.347,172.2272,-8.3691,0.0000
C01138=-19.200,-90.783,31.942,177.6276,-3.1482,0.0000
C01139=-20.718,-92.664,32.394,179.6431,-0.3988,0.0000
C01140=-22.602,-94.262,32.617,-179.9322,0.0374,0.0000
C01141=-25.531,-95.180,32.735,-179.6818,0.0477,0.0000
C01142=-29.149,-95.246,32.831,-179.3160,-0.0705,0.0000
C01143=-32.878,-94.386,32.928,-179.9997,-0.0001,0.0000
C01144=-36.490,-93.098,32.991,-179.9988,-0.0004,0.0000
C01145=-40.028,-91.633,32.991,-179.9989,-0.0005,0.0000
C01146=-43.493,-89.989,32.928,-179.9997,-0.0001,0.0000
C01147=-46.737,-87.960,32.831,-179.4665,-0.4338,0.0000
C01148=-49.249,-85.356,32.735,-179.8087,-0.2587,0.0000
C01149=-50.671,-82.635,32.617,-179.9785,-0.0744,0.0000
C01150=-50.874,-80.174,32.394,-179.9703,0.5344,0.0000
C01151=-50.617,-77.770,31.942,-179.4502,3.9008,0.0000
C01152=-50.455,-75.506,31.347,-179.5699,11.3401,0.0000
C01153=-50.836,-73.375,30.762,173.8456,22.5147,0.0000
C01154=-52.312,-71.113,30.332,157.4247,26.4448,0.0000
C01155=-55.379,-68.290,30.160,152.2123,24.6497,0.0000
C01156=-58.753,-65.381,30.152,152.3768,25.0757,0.0000
C01157=-62.157,-62.157,30.157,153.6112,26.3893,0.0000
C01158=-65.381,-58.753,30.152,154.9239,27.6229,0.0000
C01159=-68.290,-55.379,30.160,155.3497,27.7869,0.0000
C01160=-71.113,-52.312,30.332,153.5556,22.5759,0.0000
C01161=-73.375,-50.836,30.762,157.4853,6.1544,0.0000
C01162=-75.506,-50.455,31.347,168.6599,-0.4301,0.0000
C01163=-77.770,-50.617,31.942,176.0992,-0.5498,0.0000
C01164=-80.174,-50.874,32.394,179.4656,-0.0297,0.0000
C01165=-82.635,-50.671,32.617,-179.9256,-0.0215,0.0000
C01166=-85.356,-49.249,32.735,-179.7413,-0.1913,0.0000
C01167=-87.960,-46.737,32.831,-179.5662,-0.5335,0.0000
C01168=-89.989,-43.493,32.928,-179.9999,-0.0003,0.0000
C01169=-91.633,-40.028,32.991,-179.9995,-0.0011,0.0000
C01170=-93.098,-36.490,32.991,-179.9996,-0.0012,0.0000
C01171=-94.386,-32.878,32.928,-179.9999,-0.0003,0.0000
C01172=-95.246,-29.149,32.831,-179.9295,-0.6840,0.0000
C01173=-95.180,-25.531,32.735,179.9523,-0.3182,0.0000
C01174=-94.262,-22.602,32.617,179.9626,-0.0678,0.0000
C01175=-92.664,-20.718,32.394,-179.6012,0.3569,0.0000
C01176=-90.783,-19.200,31.942,-176.8518,2.3724,0.0000
C01177=-89.068,-17.714,31.347,-171.6309,7.7728,0.0000
C01178=-87.830,-15.938,30.762,-167.7644,20.2718,0.0000
C01179=-87.274,-13.294,30.332,-176.6967,32.8496,0.0000
C01180=-87.447,-9.129,30.160,177.2439,34.8804,0.0000
C01181=-87.776,-4.687,30.152,177.7573,35.0266,0.0000
C01182=-87.904,0.000,30.157,-179.9996,35.0568,0.0000
C01183=-87.776,4.687,30.152,-177.7578,35.0266,0.0000
C01184=-87.447,9.130,30.160,-177.2451,34.8803,0.0000
C01185=-87.274,13.294,30.332,176.6975,32.8497,0.0000
C01186=-87.830,15.938,30.762,167.7644,20.2718,0.0000
C01187=-89.068,17.714,31.347,171.6309,7.7728,0.0000
C01188=-90.783,19.200,31.942,176.8518,2.3724,0.0000
C01189=-92.664,20.718,32.394,179.6012,0.3569,0.0000
C01190=-94.262,22.602,32.617,-179.9626,-0.0678,0.0000
C01191=-95.180,25.531,32.735,-179.9523,-0.3182,0.0000
C01192=-95.246,29.149,32.831,179.9295,-0.6840,0.0000
C01193=-94.386,32.878,32.928,179.9999,-0.0003,0.0000
C01194=-93.098,36.490,32.991,179.9996,-0.0012,0.0000
C01195=-91.633,40.028,32.991,179.9995,-0.0011,0.0000
C01196=-89.989,43.493,32.928,179.9999,-0.0003,0.0000
C01197=-87.960,46.737,32.831,179.5662,-0.5335,0.0000
C01198=-85.356,49.249,32.735,179.7413,-0.1913,0.0000
C01199=-82.635,50.671,32.617,179.9256,-0.0215,0.0000
C01200=-80.174,50.874,32.394,-179.4656,-0.0297,0.0000
C01201=-77.770,50.617,31.942,-176.0992,-0.5498,0.0000
C01202=-75.506,50.455,31.347,-168.6599,-0.4301,0.0000
C01203=-73.375,50.836,30.762,-157.4853,6.1544,0.0000
C01204=-71.113,52.312,30.332,-153.5552,22.5753,0.0000
C01205=-68.290,55.379,30.160,-155.3503,27.7877,0.0000
C01206=-65.381,58.753,30.152,-154.9243,27.6232,0.0000
C01207=-62.157,62.157,30.157,-153.6107,26.3888,0.0000
C01208=-58.753,65.381,30.152,-152.3771,25.0761,0.0000
C01209=-55.379,68.290,30.160,-152.2131,24.6503,0.0000
C01210=-52.312,71.113,30.332,-157.4241,26.4444,0.0000
C01211=-50.836,73.375,30.762,-173.8456,22.5147,0.0000
C01212=-50.455,75.506,31.347,179.5699,11.3401,0.0000
C01213=-50.617,77.770,31.942,179.4502,3.9008,0.0000
C01214=-50.874,80.174,32.394,179.9703,0.5344,0.0000
C01215=-50.671,82.635,32.617,179.9785,-0.0744,0.0000
C01216=-49.249,85.356,32.735,179.8087,-0.2587,0.0000
C01217=-46.737,87.960,32.831,179.4665,-0.4338,0.0000
C01218=-43.493,89.989,32.928,179.9997,-0.0001,0.0000
C01219=-40.028,91.633,32.991,179.9989,-0.0005,0.0000
C01220=-36.490,93.098,32.991,179.9988,-0.0004,0.0000
C01221=-32.878,94.386,32.928,179.9997,-0.0001,0.0000
C01222=-29.149,95.246,32.831,179.3160,-0.0705,0.0000
C01223=-25.531,95.180,32.735,179.6818,0.0477,0.0000
C01224=-22.602,94.262,32.617,179.9322,0.0374,0.0000
C01225=-20.718,92.664,32.394,-179.6431,-0.3988,0.0000
C01226=-19.200,90.783,31.942,-177.6276,-3.1482,0.0000
C01227=-17.714,89.068,31.347,-172.2272,-8.3691,0.0000
C01228=-15.938,87.830,30.762,-159.7282,-12.2356,0.0000
C01229=-13.294,87.274,30.332,-147.1503,-3.3025,0.0000
C01230=-9.130,87.447,30.160,-145.1197,2.7549,0.0000
C01231=-4.687,87.776,30.152,-144.9734,2.2422,0.0000
C01232=0.000,87.904,30.157,-144.9432,0.0004,0.0000
C01233=0.000,86.627,31.948,-144.1028,0.0004,0.0000
C01234=4.570,86.503,31.943,-144.1331,-2.3009,0.0000
C01235=8.933,86.186,31.951,-144.2840,-2.6354,0.0000
C01236=13.053,86.053,32.146,-146.6498,4.4571,0.0000
C01237=15.641,86.712,32.633,-161.4230,13.0408,0.0000
C01238=17.370,88.113,33.299,-173.7884,7.6720,0.0000
C01239=18.822,90.045,33.980,-178.5738,2.1633,0.0000
C01240=20.308,92.176,34.500,179.5624,-0.5662,0.0000
C01241=22.152,94.017,34.757,179.0872,-0.5942,0.0000
C01242=25.107,95.129,34.893,179.2076,-0.1524,0.0000
C01243=28.812,95.307,35.004,179.1192,0.0737,0.0000
C01244=32.664,94.457,35.116,179.9841,0.0052,0.0000
C01245=36.417,93.126,35.190,179.9970,0.0012,0.0000
C01246=40.099,91.601,35.190,179.9971,0.0013,0.0000
C01247=43.694,89.888,35.116,179.9851,0.0076,0.0000
C01248=47.019,87.765,35.004,179.3251,0.5708,0.0000
C01249=49.513,85.019,34.893,179.5474,0.6681,0.0000
C01250=50.816,82.144,34.757,179.7747,1.0655,0.0000
C01251=50.818,79.538,34.500,-179.9091,0.7097,0.0000
C01252=50.362,76.980,33.980,179.4783,-2.5374,0.0000
C01253=50.022,74.588,33.299,178.9521,-9.7713,0.0000
C01254=50.255,72.374,32.633,-175.7750,-21.8720,0.0000
C01255=51.619,70.079,32.146,-157.6940,-27.4964,0.0000
C01256=54.626,67.259,31.951,-151.5886,-25.4479,0.0000
C01257=57.935,64.399,31.943,-151.6465,-25.7724,0.0000
C01258=61.254,61.254,31.948,-152.8966,-27.1039,0.0000
C01259=64.398,57.936,31.943,-154.2272,-28.3532,0.0000
C01260=67.259,54.626,31.951,-154.5515,-28.4105,0.0000
C01261=70.079,51.619,32.146,-152.5039,-22.3066,0.0000
C01262=72.374,50.255,32.633,-158.1280,-4.2250,0.0000
C01263=74.588,50.022,33.299,-170.2287,1.0479,0.0000
C01264=76.980,50.362,33.980,-177.4626,0.5217,0.0000
C01265=79.538,50.818,34.500,179.2903,-0.0909,0.0000
C01266=82.144,50.816,34.757,178.9345,0.2253,0.0000
C01267=85.019,49.513,34.893,179.3319,0.4526,0.0000
C01268=87.765,47.019,35.004,179.4292,0.6749,0.0000
C01269=89.888,43.694,35.116,179.9924,0.0149,0.0000
C01270=91.601,40.099,35.190,179.9987,0.0029,0.0000
C01271=93.126,36.417,35.190,179.9988,0.0030,0.0000
C01272=94.457,32.664,35.116,179.9948,0.0159,0.0000
C01273=95.307,28.812,35.004,179.9263,0.8808,0.0000
C01274=95.129,25.107,34.893,-179.8476,0.7924,0.0000
C01275=94.017,22.152,34.757,-179.4058,0.9128,0.0000
C01276=92.176,20.308,34.500,-179.4338,0.4376,0.0000
C01277=90.045,18.822,33.980,177.8367,-1.4262,0.0000
C01278=88.113,17.370,33.299,172.3280,-6.2116,0.0000
C01279=86.712,15.641,32.633,166.9592,-18.5770,0.0000
C01280=86.053,13.053,32.146,175.5429,-33.3502,0.0000
C01281=86.186,8.933,31.951,-177.3646,-35.7160,0.0000
C01282=86.503,4.570,31.943,-177.6991,-35.8669,0.0000
C01283=86.627,0.000,31.948,179.9996,-35.8972,0.0000
C01284=86.503,-4.570,31.943,177.6997,-35.8669,0.0000
C01285=86.186,-8.933,31.951,177.3659,-35.7159,0.0000
C01286=86.053,-13.053,32.146,-175.5437,-33.3504,0.0000
C01287=86.712,-15.641,32.633,-166.9592,-18.5770,0.0000
C01288=88.113,-17.370,33.299,-172.3280,-6.2116,0.0000
C01289=90.045,-18.822,33.980,-177.8367,-1.4262,0.0000
C01290=92.176,-20.308,34.500,179.4338,0.4376,0.0000
C01291=94.017,-22.152,34.757,179.4058,0.9128,0.0000
C01292=95.129,-25.107,34.893,179.8476,0.7924,0.0000
C01293=95.307,-28.812,35.004,-179.9263,0.8808,0.0000
C01294=94.457,-32.664,35.116,-179.9948,0.0159,0.0000
C01295=93.126,-36.417,35.190,-179.9988,0.0030,0.0000
C01296=91.601,-40.099,35.190,-179.9987,0.0029,0.0000
C01297=89.888,-43.694,35.116,-179.9924,0.0149,0.0000
C01298=87.765,-47.019,35.004,-179.4292,0.6749,0.0000
C01299=85.019,-49.513,34.893,-179.3319,0.4526,0.0000
C01300=82.144,-50.816,34.757,-178.9345,0.2253,0.0000
C01301=79.538,-50.818,34.500,-179.2903,-0.0909,0.0000
C01302=76.980,-50.362,33.980,177.4626,0.5217,0.0000
C01303=74.588,-50.022,33.299,170.2287,1.0479,0.0000
C01304=72.374,-50.255,32.633,158.1280,-4.2250,0.0000
C01305=70.079,-51.619,32.146,152.5036,-22.3060,0.0000
C01306=67.259,-54.626,31.951,154.5521,-28.4114,0.0000
C01307=64.399,-57.935,31.943,154.2276,-28.3535,0.0000
C01308=61.254,-61.254,31.948,152.8961,-27.1034,0.0000
C01309=57.936,-64.398,31.943,151.6468,-25.7728,0.0000
C01310=54.626,-67.259,31.951,151.5895,-25.4485,0.0000
C01311=51.619,-70.079,32.146,157.6934,-27.4961,0.0000
C01312=50.255,-72.374,32.633,175.7750,-21.8720,0.0000
C01313=50.022,-74.588,33.299,-178.9521,-9.7713,0.0000
C01314=50.362,-76.980,33.980,-179.4783,-2.5374,0.0000
C01315=50.818,-79.538,34.500,179.9091,0.7097,0.0000
C01316=50.816,-82.144,34.757,-179.7747,1.0655,0.0000
C01317=49.513,-85.019,34.893,-179.5474,0.6681,0.0000
C01318=47.019,-87.765,35.004,-179.3251,0.5708,0.0000
C01319=43.694,-89.888,35.116,-179.9851,0.0076,0.0000
C01320=40.099,-91.601,35.190,-179.9971,0.0013,0.0000
C01321=36.417,-93.126,35.190,-179.9970,0.0012,0.0000
C01322=32.664,-94.457,35.116,-179.9841,0.0052,0.0000
C01323=28.812,-95.307,35.004,-179.1192,0.0737,0.0000
C01324=25.107,-95.129,34.893,-179.2076,-0.1524,0.0000
C01325=22.152,-94.017,34.757,-179.0872,-0.5942,0.0000
C01326=20.308,-92.176,34.500,-179.5624,-0.5662,0.0000
C01327=18.822,-90.045,33.980,178.5738,2.1633,0.0000
C01328=17.370,-88.113,33.299,173.7884,7.6720,0.0000
C01329=15.641,-86.712,32.633,161.4230,13.0408,0.0000
C01330=13.053,-86.053,32.146,146.6498,4.4571,0.0000
C01331=8.933,-86.186,31.951,144.2840,-2.6354,0.0000
C01332=4.570,-86.503,31.943,144.1331,-2.3009,0.0000
C01333=0.000,-86.627,31.948,144.1028,0.0004,0.0000
C01334=0.000,-86.627,31.948,144.1028,0.0004,0.0000
C01335=-4.570,-86.503,31.943,144.1331,2.3003,0.0000
C01336=-8.933,-86.186,31.951,144.2841,2.6341,0.0000
C01337=-13.053,-86.053,32.146,146.6496,-4.4563,0.0000
C01338=-15.641,-86.712,32.633,161.4230,-13.0408,0.0000
C01339=-17.370,-88.113,33.299,173.7884,-7.6720,0.0000
C01340=-18.822,-90.045,33.980,178.5738,-2.1633,0.0000
C01341=-20.308,-92.176,34.500,-179.5624,0.5662,0.0000
C01342=-22.152,-94.017,34.757,-179.0872,0.5942,0.0000
C01343=-25.107,-95.129,34.893,-179.2076,0.1524,0.0000
C01344=-28.812,-95.307,35.004,-179.1192,-0.0737,0.0000
C01345=-32.664,-94.457,35.116,-179.9841,-0.0052,0.0000
C01346=-36.417,-93.126,35.190,-179.9970,-0.0012,0.0000
C01347=-40.099,-91.601,35.190,-179.9971,-0.0013,0.0000
C01348=-43.694,-89.888,35.116,-179.9851,-0.0076,0.0000
C01349=-47.019,-87.765,35.004,-179.3251,-0.5708,0.0000
C01350=-49.513,-85.019,34.893,-179.5474,-0.6681,0.0000
C01351=-50.816,-82.144,34.757,-179.7747,-1.0655,0.0000
C01352=-50.818,-79.538,34.500,179.9091,-0.7097,0.0000
C01353=-50.362,-76.980,33.980,-179.4783,2.5374,0.0000
C01354=-50.022,-74.588,33.299,-178.9521,9.7713,0.0000
C01355=-50.255,-72.374,32.633,175.7750,21.8720,0.0000
C01356=-51.619,-70.079,32.146,157.6940,27.4964,0.0000
C01357=-54.626,-67.259,31.951,151.5886,25.4479,0.0000
C01358=-57.935,-64.399,31.943,151.6465,25.7724,0.0000
C01359=-61.254,-61.254,31.948,152.8966,27.1039,0.0000
C01360=-64.398,-57.936,31.943,154.2272,28.3532,0.0000
C01361=-67.259,-54.626,31.951,154.5515,28.4105,0.0000
C01362=-70.079,-51.619,32.146,152.5039,22.3066,0.0000
C01363=-72.374,-50.255,32.633,158.1280,4.2250,0.0000
C01364=-74.588,-50.022,33.299,170.2287,-1.0479,0.0000
C01365=-76.980,-50.362,33.980,177.4626,-0.5217,0.0000
C01366=-79.538,-50.818,34.500,-179.2903,0.0909,0.0000
C01367=-82.144,-50.816,34.757,-178.9345,-0.2253,0.0000
C01368=-85.019,-49.513,34.893,-179.3319,-0.4526,0.0000
C01369=-87.765,-47.019,35.004,-179.4292,-0.6749,0.0000
C01370=-89.888,-43.694,35.116,-179.9924,-0.0149,0.0000
C01371=-91.601,-40.099,35.190,-179.9987,-0.0029,0.0000
C01372=-93.126,-36.417,35.190,-179.9988,-0.0030,0.0000
C01373=-94.457,-32.664,35.116,-179.9948,-0.0159,0.0000
C01374=-95.307,-28.812,35.004,-179.9263,-0.8808,0.0000
C01375=-95.129,-25.107,34.893,179.8476,-0.7924,0.0000
C01376=-94.017,-22.152,34.757,179.4058,-0.9128,0.0000
C01377=-92.176,-20.308,34.500,179.4338,-0.4376,0.0000
C01378=-90.045,-18.822,33.980,-177.8367,1.4262,0.0000
C01379=-88.113,-17.370,33.299,-172.3280,6.2116,0.0000
C01380=-86.712,-15.641,32.633,-166.9592,18.5770,0.0000
C01381=-86.053,-13.053,32.146,-175.5429,33.3502,0.0000
C01382=-86.186,-8.933,31.951,177.3646,35.7160,0.0000
C01383=-86.503,-4.570,31.943,177.6991,35.8669,0.0000
C01384=-86.627,0.000,31.948,-179.9996,35.8972,0.0000
C01385=-86.503,4.570,31.943,-177.6997,35.8669,0.0000
C01386=-86.186,8.933,31.951,-177.3659,35.7159,0.0000
C01387=-86.053,13.053,32.146,175.5437,33.3504,0.0000
C01388=-86.712,15.641,32.633,166.9592,18.5770,0.0000
C01389=-88.113,17.370,33.299,172.3280,6.2116,0.0000
C01390=-90.045,18.822,33.980,177.8367,1.4262,0.0000
C01391=-92.176,20.308,34.500,-179.4338,-0.4376,0.0000
C01392=-94.017,22.152,34.757,-179.4058,-0.9128,0.0000
C01393=-95.129,25.107,34.893,-179.8476,-0.7924,0.0000
C01394=-95.307,28.812,35.004,179.9263,-0.8808,0.0000
C01395=-94.457,32.664,35.116,179.9948,-0.0159,0.0000
C01396=-93.126,36.417,35.190,179.9988,-0.0030,0.0000
C01397=-91.601,40.099,35.190,179.9987,-0.0029,0.0000
C01398=-89.888,43.694,35.116,179.9924,-0.0149,0.0000
C01399=-87.765,47.019,35.004,179.4292,-0.6749,0.0000
C01400=-85.019,49.513,34.893,179.3319,-0.4526,0.0000
C01401=-82.144,50.816,34.757,178.9345,-0.2253,0.0000
C01402=-79.538,50.818,34.500,179.2903,0.0909,0.0000
C01403=-76.980,50.362,33.980,-177.4626,-0.5217,0.0000
C01404=-74.588,50.022,33.299,-170.2287,-1.0479,0.0000
C01405=-72.374,50.255,32.633,-158.1280,4.2250,0.0000
C01406=-70.079,51.619,32.146,-152.5036,22.3060,0.0000
C01407=-67.259,54.626,31.951,-154.5521,28.4114,0.0000
C01408=-64.399,57.935,31.943,-154.2276,28.3535,0.0000
C01409=-61.254,61.254,31.948,-152.8961,27.1034,0.0000
C01410=-57.936,64.398,31.943,-151.6468,25.7728,0.0000
C01411=-54.626,67.259,31.951,-151.5895,25.4485,0.0000
C01412=-51.619,70.079,32.146,-157.6934,27.4961,0.0000
C01413=-50.255,72.374,32.633,-175.7750,21.8720,0.0000
C01414=-50.022,74.588,33.299,178.9521,9.7713,0.0000
C01415=-50.362,76.980,33.980,179.4783,2.5374,0.0000
C01416=-50.818,79.538,34.500,-179.9091,-0.7097,0.0000
C01417=-50.816,82.144,34.757,179.7747,-1.0655,0.0000
C01418=-49.513,85.019,34.893,179.5474,-0.6681,0.0000
C01419=-47.019,87.765,35.004,179.3251,-0.5708,0.0000
C01420=-43.694,89.888,35.116,179.9851,-0.0076,0.0000
C01421=-40.099,91.601,35.190,179.9971,-0.0013,0.0000
C01422=-36.417,93.126,35.190,179.9970,-0.0012,0.0000
C01423=-32.664,94.457,35.116,179.9841,-0.0052,0.0000
C01424=-28.812,95.307,35.004,179.1192,-0.0737,0.0000
C01425=-25.107,95.129,34.893,179.2076,0.1524,0.0000
C01426=-22.152,94.017,34.757,179.0872,0.5942,0.0000
C01427=-20.308,92.176,34.500,179.5624,0.5662,0.0000
C01428=-18.822,90.045,33.980,-178.5738,-2.1633,0.0000
C01429=-17.370,88.113,33.299,-173.7884,-7.6720,0.0000
C01430=-15.641,86.712,32.633,-161.4230,-13.0408,0.0000
C01431=-13.053,86.053,32.146,-146.6496,-4.4563,0.0000
C01432=-8.933,86.186,31.951,-144.2841,2.6341,0.0000
C01433=-4.570,86.503,31.943,-144.1331,2.3003,0.0000
C01434=0.000,86.627,31.948,-144.1028,0.0004,0.0000
C01435=0.000,85.325,33.722,-143.3716,0.0004,0.0000
C01436=4.451,85.206,33.716,-143.4019,-2.3496,0.0000
C01437=8.733,84.900,33.725,-143.5590,-2.4835,0.0000
C01438=12.808,84.808,33.943,-146.3185,5.6572,0.0000
C01439=15.338,85.570,34.490,-163.2997,13.4594,0.0000
C01440=17.019,87.137,35.239,-175.1574,6.7892,0.0000
C01441=18.435,89.289,36.009,-179.3291,1.1505,0.0000
C01442=19.887,91.675,36.600,178.9476,-1.5568,0.0000
C01443=21.692,93.766,36.894,178.3326,-1.2566,0.0000
C01444=24.671,95.076,37.049,178.7354,-0.2964,0.0000
C01445=28.465,95.370,37.176,178.9222,0.0699,0.0000
C01446=32.445,94.529,37.304,179.9684,0.0102,0.0000
C01447=36.342,93.155,37.389,179.9952,0.0018,0.0000
C01448=40.172,91.569,37.389,179.9953,0.0021,0.0000
C01449=43.901,89.784,37.304,179.9704,0.0151,0.0000
C01450=47.309,87.565,37.176,179.1885,0.7127,0.0000
C01451=49.784,84.674,37.049,179.3153,1.1038,0.0000
C01452=50.965,81.641,36.894,179.7094,2.0671,0.0000
C01453=50.762,78.886,36.600,-179.6431,1.8447,0.0000
C01454=50.101,76.172,36.009,179.6608,-1.2879,0.0000
C01455=49.580,73.649,35.239,178.6093,-8.1993,0.0000
C01456=49.662,71.353,34.490,-177.5427,-20.8758,0.0000
C01457=50.912,69.025,33.943,-158.1390,-28.4266,0.0000
C01458=53.858,66.209,33.725,-151.0673,-26.1712,0.0000
C01459=57.102,63.397,33.716,-151.0082,-26.3858,0.0000
C01460=60.334,60.334,33.722,-152.2699,-27.7306,0.0000
C01461=63.397,57.102,33.716,-153.6139,-28.9915,0.0000
C01462=66.209,53.858,33.725,-153.8281,-28.9318,0.0000
C01463=69.025,50.912,33.943,-151.5737,-21.8617,0.0000
C01464=71.353,49.662,34.490,-159.1242,-2.4573,0.0000
C01465=73.649,49.580,35.239,-171.8007,1.3907,0.0000
C01466=76.172,50.101,36.009,-178.7121,0.3392,0.0000
C01467=78.886,50.762,36.600,178.1553,-0.3569,0.0000
C01468=81.641,50.965,36.894,177.9329,0.2906,0.0000
C01469=84.674,49.784,37.049,178.8962,0.6847,0.0000
C01470=87.565,47.309,37.176,179.2873,0.8115,0.0000
C01471=89.784,43.901,37.304,179.9849,0.0296,0.0000
C01472=91.569,40.172,37.389,179.9979,0.0047,0.0000
C01473=93.155,36.342,37.389,179.9982,0.0048,0.0000
C01474=94.529,32.445,37.304,179.9898,0.0316,0.0000
C01475=95.370,28.465,37.176,179.9301,1.0778,0.0000
C01476=95.076,24.671,37.049,-179.7036,1.2646,0.0000
C01477=93.766,21.692,36.894,-178.7434,1.6674,0.0000
C01478=91.675,19.887,36.600,-178.4432,1.0524,0.0000
C01479=89.289,18.435,36.009,178.8495,-0.6709,0.0000
C01480=87.137,17.019,35.239,173.2108,-4.8426,0.0000
C01481=85.570,15.338,34.490,166.5406,-16.7003,0.0000
C01482=84.808,12.808,33.943,174.3428,-33.6815,0.0000
C01483=84.900,8.733,33.725,-177.5165,-36.4410,0.0000
C01484=85.206,4.451,33.716,-177.6504,-36.5981,0.0000
C01485=85.325,0.000,33.722,179.9996,-36.6284,0.0000
C01486=85.206,-4.451,33.716,177.6510,-36.5982,0.0000
C01487=84.900,-8.733,33.725,177.5180,-36.4409,0.0000
C01488=84.808,-12.808,33.943,-174.3436,-33.6818,0.0000
C01489=85.570,-15.338,34.490,-166.5406,-16.7003,0.0000
C01490=87.137,-17.019,35.239,-173.2108,-4.8426,0.0000
C01491=89.289,-18.435,36.009,-178.8495,-0.6709,0.0000
C01492=91.675,-19.887,36.600,178.4432,1.0524,0.0000
C01493=93.766,-21.692,36.894,178.7434,1.6674,0.0000
C01494=95.076,-24.671,37.049,179.7036,1.2646,0.0000
C01495=95.370,-28.465,37.176,-179.9301,1.0778,0.0000
C01496=94.529,-32.445,37.304,-179.9898,0.0316,0.0000
C01497=93.155,-36.342,37.389,-179.9982,0.0048,0.0000
C01498=91.569,-40.172,37.389,-179.9979,0.0047,0.0000
C01499=89.784,-43.901,37.304,-179.9849,0.0296,0.0000
C01500=87.565,-47.309,37.176,-179.2873,0.8115,0.0000
C01501=84.674,-49.784,37.049,-178.8962,0.6847,0.0000
C01502=81.641,-50.965,36.894,-177.9329,0.2906,0.0000
C01503=78.886,-50.762,36.600,-178.1553,-0.3569,0.0000
C01504=76.172,-50.101,36.009,178.7121,0.3392,0.0000
C01505=73.649,-49.580,35.239,171.8007,1.3907,0.0000
C01506=71.353,-49.662,34.490,159.1242,-2.4573,0.0000
C01507=69.025,-50.912,33.943,151.5734,-21.8610,0.0000
C01508=66.209,-53.858,33.725,153.8288,-28.9327,0.0000
C01509=63.397,-57.102,33.716,153.6142,-28.9918,0.0000
C01510=60.334,-60.334,33.722,152.2694,-27.7301,0.0000
C01511=57.102,-63.397,33.716,151.0085,-26.3861,0.0000
C01512=53.858,-66.209,33.725,151.0682,-26.1719,0.0000
C01513=50.912,-69.025,33.943,158.1383,-28.4263,0.0000
C01514=49.662,-71.353,34.490,177.5427,-20.8758,0.0000
C01515=49.580,-73.649,35.239,-178.6093,-8.1993,0.0000
C01516=50.101,-76.172,36.009,-179.6608,-1.2879,0.0000
C01517=50.762,-78.886,36.600,179.6431,1.8447,0.0000
C01518=50.965,-81.641,36.894,-179.7094,2.0671,0.0000
C01519=49.784,-84.674,37.049,-179.3153,1.1038,0.0000
C01520=47.309,-87.565,37.176,-179.1885,0.7127,0.0000
C01521=43.901,-89.784,37.304,-179.9704,0.0151,0.0000
C01522=40.172,-91.569,37.389,-179.9953,0.0021,0.0000
C01523=36.342,-93.155,37.389,-179.9952,0.0018,0.0000
C01524=32.445,-94.529,37.304,-179.9684,0.0102,0.0000
C01525=28.465,-95.370,37.176,-178.9222,0.0699,0.0000
C01526=24.671,-95.076,37.049,-178.7354,-0.2964,0.0000
C01527=21.692,-93.766,36.894,-178.3326,-1.2566,0.0000
C01528=19.887,-91.675,36.600,-178.9476,-1.5568,0.0000
C01529=18.435,-89.289,36.009,179.3291,1.1505,0.0000
C01530=17.019,-87.137,35.239,175.1574,6.7892,0.0000
C01531=15.338,-85.570,34.490,163.2997,13.4594,0.0000
C01532=12.808,-84.808,33.943,146.3185,5.6572,0.0000
C01533=8.733,-84.900,33.725,143.5590,-2.4835,0.0000
C01534=4.451,-85.206,33.716,143.4019,-2.3496,0.0000
C01535=0.000,-85.325,33.722,143.3716,0.0004,0.0000
C01536=0.000,-85.325,33.722,143.3716,0.0004,0.0000
C01537=-4.451,-85.206,33.716,143.4018,2.3490,0.0000
C01538=-8.733,-84.900,33.725,143.5591,2.4820,0.0000
C01539=-12.808,-84.808,33.943,146.3182,-5.6564,0.0000
C01540=-15.338,-85.570,34.490,163.2997,-13.4594,0.0000
C01541=-17.019,-87.137,35.239,175.1574,-6.7892,0.0000
C01542=-18.435,-89.289,36.009,179.3291,-1.1505,0.0000
C01543=-19.887,-91.675,36.600,-178.9476,1.5568,0.0000
C01544=-21.692,-93.766,36.894,-178.3326,1.2566,0.0000
C01545=-24.671,-95.076,37.049,-178.7354,0.2964,0.0000
C01546=-28.465,-95.370,37.176,-178.9222,-0.0699,0.0000
C01547=-32.445,-94.529,37.304,-179.9684,-0.0102,0.0000
C01548=-36.342,-93.155,37.389,-179.9952,-0.0018,0.0000
C01549=-40.172,-91.569,37.389,-179.9953,-0.0021,0.0000
C01550=-43.901,-89.784,37.304,-179.9704,-0.0151,0.0000
C01551=-47.309,-87.565,37.176,-179.1885,-0.7127,0.0000
C01552=-49.784,-84.674,37.049,-179.3153,-1.1038,0.0000
C01553=-50.965,-81.641,36.894,-179.7094,-2.0671,0.0000
C01554=-50.762,-78.886,36.600,179.6431,-1.8447,0.0000
C01555=-50.101,-76.172,36.009,-179.6608,1.2879,0.0000
C01556=-49.580,-73.649,35.239,-178.6093,8.1993,0.0000
C01557=-49.662,-71.353,34.490,177.5427,20.8758,0.0000
C01558=-50.912,-69.025,33.943,158.1390,28.4266,0.0000
C01559=-53.858,-66.209,33.725,151.0673,26.1712,0.0000
C01560=-57.102,-63.397,33.716,151.0082,26.3858,0.0000
C01561=-60.334,-60.334,33.722,152.2699,27.7306,0.0000
C01562=-63.397,-57.102,33.716,153.6139,28.9915,0.0000
C01563=-66.209,-53.858,33.725,153.8281,28.9318,0.0000
C01564=-69.025,-50.912,33.943,151.5737,21.8617,0.0000
C01565=-71.353,-49.662,34.490,159.1242,2.4573,0.0000
C01566=-73.649,-49.580,35.239,171.8007,-1.3907,0.0000
C01567=-76.172,-50.101,36.009,178.7121,-0.3392,0.0000
C01568=-78.886,-50.762,36.600,-178.1553,0.3569,0.0000
C01569=-81.641,-50.965,36.894,-177.9329,-0.2906,0.0000
C01570=-84.674,-49.784,37.049,-178.8962,-0.6847,0.0000
C01571=-87.565,-47.309,37.176,-179.2873,-0.8115,0.0000
C01572=-89.784,-43.901,37.304,-179.9849,-0.0296,0.0000
C01573=-91.569,-40.172,37.389,-179.9979,-0.0047,0.0000
C01574=-93.155,-36.342,37.389,-179.9982,-0.0048,0.0000
C01575=-94.529,-32.445,37.304,-179.9898,-0.0316,0.0000
C01576=-95.370,-28.465,37.176,-179.9301,-1.0778,0.0000
C01577=-95.076,-24.671,37.049,179.7036,-1.2646,0.0000
C01578=-93.766,-21.692,36.894,178.7434,-1.6674,0.0000
C01579=-91.675,-19.887,36.600,178.4432,-1.0524,0.0000
C01580=-89.289,-18.435,36.009,-178.8495,0.6709,0.0000
C01581=-87.137,-17.019,35.239,-173.2108,4.8426,0.0000
C01582=-85.570,-15.338,34.490,-166.5406,16.7003,0.0000
C01583=-84.808,-12.808,33.943,-174.3428,33.6815,0.0000
C01584=-84.900,-8.733,33.725,177.5165,36.4410,0.0000
C01585=-85.206,-4.451,33.716,177.6504,36.5981,0.0000
C01586=-85.325,0.000,33.722,-179.9996,36.6284,0.0000
C01587=-85.206,4.451,33.716,-177.6510,36.5982,0.0000
C01588=-84.900,8.733,33.725,-177.5180,36.4409,0.0000
C01589=-84.808,12.808,33.943,174.3436,33.6818,0.0000
C01590=-85.570,15.338,34.490,166.5406,16.7003,0.0000
C01591=-87.137,17.019,35.239,173.2108,4.8426,0.0000
C01592=-89.289,18.435,36.009,178.8495,0.6709,0.0000
C01593=-91.675,19.887,36.600,-178.4432,-1.0524,0.0000
C01594=-93.766,21.692,36.894,-178.7434,-1.6674,0.0000
C01595=-95.076,24.671,37.049,-179.7036,-1.2646,0.0000
C01596=-95.370,28.465,37.176,179.9301,-1.0778,0.0000
C01597=-94.529,32.445,37.304,179.9898,-0.0316,0.0000
C01598=-93.155,36.342,37.389,179.9982,-0.0048,0.0000
C01599=-91.569,40.172,37.389,179.9979,-0.0047,0.0000
C01600=-89.784,43.901,37.304,179.9849,-0.0296,0.0000
C01601=-87.565,47.309,37.176,179.2873,-0.8115,0.0000
C01602=-84.674,49.784,37.049,178.8962,-0.6847,0.0000
C01603=-81.641,50.965,36.894,177.9329,-0.2906,0.0000
C01604=-78.886,50.762,36.600,178.1553,0.3569,0.0000
C01605=-76.172,50.101,36.009,-178.7121,-0.3392,0.0000
C01606=-73.649,49.580,35.239,-171.8007,-1.3907,0.0000
C01607=-71.353,49.662,34.490,-159.1242,2.4573,0.0000
C01608=-69.025,50.912,33.943,-151.5734,21.8610,0.0000
C01609=-66.209,53.858,33.725,-153.8288,28.9327,0.0000
C01610=-63.397,57.102,33.716,-153.6142,28.9918,0.0000
C01611=-60.334,60.334,33.722,-152.2694,27.7301,0.0000
C01612=-57.102,63.397,33.716,-151.0085,26.3861,0.0000
C01613=-53.858,66.209,33.725,-151.0682,26.1719,0.0000
C01614=-50.912,69.025,33.943,-158.1383,28.4263,0.0000
C01615=-49.662,71.353,34.490,-177.5427,20.8758,0.0000
C01616=-49.580,73.649,35.239,178.6093,8.1993,0.0000
C01617=-50.101,76.172,36.009,179.6608,1.2879,0.0000
C01618=-50.762,78.886,36.600,-179.6431,-1.8447,0.0000
C01619=-50.965,81.641,36.894,179.7094,-2.0671,0.0000
C01620=-49.784,84.674,37.049,179.3153,-1.1038,0.0000
C01621=-47.309,87.565,37.176,179.1885,-0.7127,0.0000
C01622=-43.901,89.784,37.304,179.9704,-0.0151,0.0000
C01623=-40.172,91.569,37.389,179.9953,-0.0021,0.0000
C01624=-36.342,93.155,37.389,179.9952,-0.0018,0.0000
C01625=-32.445,94.529,37.304,179.9684,-0.0102,0.0000
C01626=-28.465,95.370,37.176,178.9222,-0.0699,0.0000
C01627=-24.671,95.076,37.049,178.7354,0.2964,0.0000
C01628=-21.692,93.766,36.894,178.3326,1.2566,0.0000
C01629=-19.887,91.675,36.600,178.9476,1.5568,0.0000
C01630=-18.435,89.289,36.009,-179.3291,-1.1505,0.0000
C01631=-17.019,87.137,35.239,-175.1574,-6.7892,0.0000
C01632=-15.338,85.570,34.490,-163.2997,-13.4594,0.0000
C01633=-12.808,84.808,33.943,-146.3182,-5.6564,0.0000
C01634=-8.733,84.900,33.725,-143.5591,2.4820,0.0000
C01635=-4.451,85.206,33.716,-143.4018,2.3490,0.0000
C01636=0.000,85.325,33.722,-143.3716,0.0004,0.0000
C01637=0.000,84.003,35.480,-142.7415,0.0004,0.0000
C01638=4.330,83.888,35.473,-142.7716,-2.3891,0.0000
C01639=8.530,83.594,35.484,-142.9366,-2.3020,0.0000
C01640=12.558,83.543,35.726,-146.1518,6.8812,0.0000
C01641=15.030,84.409,36.333,-165.2581,13.5086,0.0000
C01642=16.662,86.143,37.169,-176.3239,5.7975,0.0000
C01643=18.041,88.518,38.031,-179.9182,0.1571,0.0000
C01644=19.458,91.164,38.697,178.4928,-2.5231,0.0000
C01645=21.221,93.510,39.027,177.6909,-1.9849,0.0000
C01646=24.227,95.023,39.203,178.2776,-0.4750,0.0000
C01647=28.112,95.435,39.346,178.7289,0.0594,0.0000
C01648=32.220,94.603,39.491,179.9530,0.0151,0.0000
C01649=36.266,93.184,39.587,179.9934,0.0025,0.0000
C01650=40.247,91.535,39.587,179.9935,0.0029,0.0000
C01651=44.111,89.678,39.491,179.9560,0.0226,0.0000
C01652=47.604,87.360,39.346,179.0591,0.8569,0.0000
C01653=50.060,84.322,39.203,179.1177,1.5538,0.0000
C01654=51.116,81.128,39.027,179.7705,3.0349,0.0000
C01655=50.704,78.221,38.697,-179.2808,2.8489,0.0000
C01656=49.835,75.348,38.031,179.9468,-0.1689,0.0000
C01657=49.130,72.694,37.169,178.4898,-6.6859,0.0000
C01658=49.058,70.314,36.333,-179.0727,-19.5923,0.0000
C01659=50.194,67.954,35.726,-158.7492,-29.2297,0.0000
C01660=53.078,65.141,35.484,-150.6424,-26.8233,0.0000
C01661=56.256,62.380,35.473,-150.4564,-26.9203,0.0000
C01662=59.399,59.399,35.480,-151.7261,-28.2744,0.0000
C01663=62.380,56.256,35.473,-153.0793,-29.5434,0.0000
C01664=65.141,53.078,35.484,-153.1760,-29.3567,0.0000
C01665=67.954,50.194,35.726,-150.7705,-21.2516,0.0000
C01666=70.314,49.058,36.333,-160.4077,-0.9273,0.0000
C01667=72.694,49.130,37.169,-173.3141,1.5102,0.0000
C01668=75.348,49.835,38.031,-179.8311,0.0532,0.0000
C01669=78.221,50.704,38.697,177.1511,-0.7192,0.0000
C01670=81.128,51.116,39.027,176.9651,0.2295,0.0000
C01671=84.322,50.060,39.203,178.4462,0.8823,0.0000
C01672=87.360,47.604,39.346,179.1431,0.9409,0.0000
C01673=89.678,44.111,39.491,179.9774,0.0440,0.0000
C01674=91.535,40.247,39.587,179.9971,0.0065,0.0000
C01675=93.184,36.266,39.587,179.9975,0.0066,0.0000
C01676=94.603,32.220,39.491,179.9849,0.0470,0.0000
C01677=95.435,28.112,39.346,179.9406,1.2711,0.0000
C01678=95.023,24.227,39.203,-179.5250,1.7224,0.0000
C01679=93.510,21.221,39.027,-178.0151,2.3091,0.0000
C01680=91.164,19.458,38.697,-177.4769,1.5072,0.0000
C01681=88.518,18.041,38.031,179.8429,-0.0818,0.0000
C01682=86.143,16.662,37.169,174.2025,-3.6761,0.0000
C01683=84.409,15.030,36.333,166.4914,-14.7419,0.0000
C01684=83.543,12.558,35.726,173.1188,-33.8482,0.0000
C01685=83.594,8.530,35.484,-177.6980,-37.0634,0.0000
C01686=83.888,4.330,35.473,-177.6109,-37.2284,0.0000
C01687=84.003,0.000,35.480,179.9996,-37.2585,0.0000
C01688=83.888,-4.330,35.473,177.6115,-37.2285,0.0000
C01689=83.594,-8.530,35.484,177.6995,-37.0633,0.0000
C01690=83.543,-12.558,35.726,-173.1197,-33.8485,0.0000
C01691=84.409,-15.030,36.333,-166.4914,-14.7419,0.0000
C01692=86.143,-16.662,37.169,-174.2025,-3.6761,0.0000
C01693=88.518,-18.041,38.031,-179.8429,-0.0818,0.0000
C01694=91.164,-19.458,38.697,177.4769,1.5072,0.0000
C01695=93.510,-21.221,39.027,178.0151,2.3091,0.0000
C01696=95.023,-24.227,39.203,179.5250,1.7224,0.0000
C01697=95.435,-28.112,39.346,-179.9406,1.2711,0.0000
C01698=94.603,-32.220,39.491,-179.9849,0.0470,0.0000
C01699=93.184,-36.266,39.587,-179.9975,0.0066,0.0000
C01700=91.535,-40.247,39.587,-179.9971,0.0065,0.0000
C01701=89.678,-44.111,39.491,-179.9774,0.0440,0.0000
C01702=87.360,-47.604,39.346,-179.1431,0.9409,0.0000
C01703=84.322,-50.060,39.203,-178.4462,0.8823,0.0000
C01704=81.128,-51.116,39.027,-176.9651,0.2295,0.0000
C01705=78.221,-50.704,38.697,-177.1511,-0.7192,0.0000
C01706=75.348,-49.835,38.031,179.8311,0.0532,0.0000
C01707=72.694,-49.130,37.169,173.3141,1.5102,0.0000
C01708=70.314,-49.058,36.333,160.4077,-0.9273,0.0000
C01709=67.954,-50.194,35.726,150.7703,-21.2508,0.0000
C01710=65.141,-53.078,35.484,153.1767,-29.3576,0.0000
C01711=62.380,-56.256,35.473,153.0797,-29.5436,0.0000
C01712=59.399,-59.399,35.480,151.7256,-28.2739,0.0000
C01713=56.256,-62.380,35.473,150.4566,-26.9207,0.0000
C01714=53.078,-65.141,35.484,150.6433,-26.8240,0.0000
C01715=50.194,-67.954,35.726,158.7484,-29.2295,0.0000
C01716=49.058,-70.314,36.333,179.0727,-19.5923,0.0000
C01717=49.130,-72.694,37.169,-178.4898,-6.6859,0.0000
C01718=49.835,-75.348,38.031,-179.9468,-0.1689,0.0000
C01719=50.704,-78.221,38.697,179.2808,2.8489,0.0000
C01720=51.116,-81.128,39.027,-179.7705,3.0349,0.0000
C01721=50.060,-84.322,39.203,-179.1177,1.5538,0.0000
C01722=47.604,-87.360,39.346,-179.0591,0.8569,0.0000
C01723=44.111,-89.678,39.491,-179.9560,0.0226,0.0000
C01724=40.247,-91.535,39.587,-179.9935,0.0029,0.0000
C01725=36.266,-93.184,39.587,-179.9934,0.0025,0.0000
C01726=32.220,-94.603,39.491,-179.9530,0.0151,0.0000
C01727=28.112,-95.435,39.346,-178.7289,0.0594,0.0000
C01728=24.227,-95.023,39.203,-178.2776,-0.4750,0.0000
C01729=21.221,-93.510,39.027,-177.6909,-1.9849,0.0000
C01730=19.458,-91.164,38.697,-178.4928,-2.5231,0.0000
C01731=18.041,-88.518,38.031,179.9182,0.1571,0.0000
C01732=16.662,-86.143,37.169,176.3239,5.7975,0.0000
C01733=15.030,-84.409,36.333,165.2581,13.5086,0.0000
C01734=12.558,-83.543,35.726,146.1518,6.8812,0.0000
C01735=8.530,-83.594,35.484,142.9366,-2.3020,0.0000
C01736=4.330,-83.888,35.473,142.7716,-2.3891,0.0000
C01737=0.000,-84.003,35.480,142.7415,0.0004,0.0000
C01738=0.000,-84.003,35.480,142.7415,0.0004,0.0000
C01739=-4.330,-83.888,35.473,142.7715,2.3885,0.0000
C01740=-8.530,-83.594,35.484,142.9367,2.3005,0.0000
C01741=-12.558,-83.543,35.726,146.1515,-6.8803,0.0000
C01742=-15.030,-84.409,36.333,165.2581,-13.5086,0.0000
C01743=-16.662,-86.143,37.169,176.3239,-5.7975,0.0000
C01744=-18.041,-88.518,38.031,179.9182,-0.1571,0.0000
C01745=-19.458,-91.164,38.697,-178.4928,2.5231,0.0000
C01746=-21.221,-93.510,39.027,-177.6909,1.9849,0.0000
C01747=-24.227,-95.023,39.203,-178.2776,0.4750,0.0000
C01748=-28.112,-95.435,39.346,-178.7289,-0.0594,0.0000
C01749=-32.220,-94.603,39.491,-179.9530,-0.0151,0.0000
C01750=-36.266,-93.184,39.587,-179.9934,-0.0025,0.0000
C01751=-40.247,-91.535,39.587,-179.9935,-0.0029,0.0000
C01752=-44.111,-89.678,39.491,-179.9560,-0.0226,0.0000
C01753=-47.604,-87.360,39.346,-179.0591,-0.8569,0.0000
C01754=-50.060,-84.322,39.203,-179.1177,-1.5538,0.0000
C01755=-51.116,-81.128,39.027,-179.7705,-3.0349,0.0000
C01756=-50.704,-78.221,38.697,179.2808,-2.8489,0.0000
C01757=-49.835,-75.348,38.031,-179.9468,0.1689,0.0000
C01758=-49.130,-72.694,37.169,-178.4898,6.6859,0.0000
C01759=-49.058,-70.314,36.333,179.0727,19.5923,0.0000
C01760=-50.194,-67.954,35.726,158.7492,29.2297,0.0000
C01761=-53.078,-65.141,35.484,150.6424,26.8233,0.0000
C01762=-56.256,-62.380,35.473,150.4564,26.9203,0.0000
C01763=-59.399,-59.399,35.480,151.7261,28.2744,0.0000
C01764=-62.380,-56.256,35.473,153.0793,29.5434,0.0000
C01765=-65.141,-53.078,35.484,153.1760,29.3567,0.0000
C01766=-67.954,-50.194,35.726,150.7705,21.2516,0.0000
C01767=-70.314,-49.058,36.333,160.4077,0.9273,0.0000
C01768=-72.694,-49.130,37.169,173.3141,-1.5102,0.0000
C01769=-75.348,-49.835,38.031,179.8311,-0.0532,0.0000
C01770=-78.221,-50.704,38.697,-177.1511,0.7192,0.0000
C01771=-81.128,-51.116,39.027,-176.9651,-0.2295,0.0000
C01772=-84.322,-50.060,39.203,-178.4462,-0.8823,0.0000
C01773=-87.360,-47.604,39.346,-179.1431,-0.9409,0.0000
C01774=-89.678,-44.111,39.491,-179.9774,-0.0440,0.0000
C01775=-91.535,-40.247,39.587,-179.9971,-0.0065,0.0000
C01776=-93.184,-36.266,39.587,-179.9975,-0.0066,0.0000
C01777=-94.603,-32.220,39.491,-179.9849,-0.0470,0.0000
C01778=-95.435,-28.112,39.346,-179.9406,-1.2711,0.0000
C01779=-95.023,-24.227,39.203,179.5250,-1.7224,0.0000
C01780=-93.510,-21.221,39.027,178.0151,-2.3091,0.0000
C01781=-91.164,-19.458,38.697,177.4769,-1.5072,0.0000
C01782=-88.518,-18.041,38.031,-179.8429,0.0818,0.0000
C01783=-86.143,-16.662,37.169,-174.2025,3.6761,0.0000
C01784=-84.409,-15.030,36.333,-166.4914,14.7419,0.0000
C01785=-83.543,-12.558,35.726,-173.1188,33.8482,0.0000
C01786=-83.594,-8.530,35.484,177.6980,37.0634,0.0000
C01787=-83.888,-4.330,35.473,177.6109,37.2284,0.0000
C01788=-84.003,0.000,35.480,-179.9996,37.2585,0.0000
C01789=-83.888,4.330,35.473,-177.6115,37.2285,0.0000
C01790=-83.594,8.530,35.484,-177.6995,37.0633,0.0000
C01791=-83.543,12.558,35.726,173.1197,33.8485,0.0000
C01792=-84.409,15.030,36.333,166.4914,14.7419,0.0000
C01793=-86.143,16.662,37.169,174.2025,3.6761,0.0000
C01794=-88.518,18.041,38.031,179.8429,0.0818,0.0000
C01795=-91.164,19.458,38.697,-177.4769,-1.5072,0.0000
C01796=-93.510,21.221,39.027,-178.0151,-2.3091,0.0000
C01797=-95.023,24.227,39.203,-179.5250,-1.7224,0.0000
C01798=-95.435,28.112,39.346,179.9406,-1.2711,0.0000
C01799=-94.603,32.220,39.491,179.9849,-0.0470,0.0000
C01800=-93.184,36.266,39.587,179.9975,-0.0066,0.0000
C01801=-91.535,40.247,39.587,179.9971,-0.0065,0.0000
C01802=-89.678,44.111,39.491,179.9774,-0.0440,0.0000
C01803=-87.360,47.604,39.346,179.1431,-0.9409,0.0000
C01804=-84.322,50.060,39.203,178.4462,-0.8823,0.0000
C01805=-81.128,51.116,39.027,176.9651,-0.2295,0.0000
C01806=-78.221,50.704,38.697,177.1511,0.7192,0.0000
C01807=-75.348,49.835,38.031,-179.8311,-0.0532,0.0000
C01808=-72.694,49.130,37.169,-173.3141,-1.5102,0.0000
C01809=-70.314,49.058,36.333,-160.4077,0.9273,0.0000
C01810=-67.954,50.194,35.726,-150.7703,21.2508,0.0000
C01811=-65.141,53.078,35.484,-153.1767,29.3576,0.0000
C01812=-62.380,56.256,35.473,-153.0797,29.5436,0.0000
C01813=-59.399,59.399,35.480,-151.7256,28.2739,0.0000
C01814=-56.256,62.380,35.473,-150.4566,26.9207,0.0000
C01815=-53.078,65.141,35.484,-150.6433,26.8240,0.0000
C01816=-50.194,67.954,35.726,-158.7484,29.2295,0.0000
C01817=-49.058,70.314,36.333,-179.0727,19.5923,0.0000
C01818=-49.130,72.694,37.169,178.4898,6.6859,0.0000
C01819=-49.835,75.348,38.031,179.9468,0.1689,0.0000
C01820=-50.704,78.221,38.697,-179.2808,-2.8489,0.0000
C01821=-51.116,81.128,39.027,179.7705,-3.0349,0.0000
C01822=-50.060,84.322,39.203,179.1177,-1.5538,0.0000
C01823=-47.604,87.360,39.346,179.0591,-0.8569,0.0000
C01824=-44.111,89.678,39.491,179.9560,-0.0226,0.0000
C01825=-40.247,91.535,39.587,179.9935,-0.0029,0.0000
C01826=-36.266,93.184,39.587,179.9934,-0.0025,0.0000
C01827=-32.220,94.603,39.491,179.9530,-0.0151,0.0000
C01828=-28.112,95.435,39.346,178.7289,-0.0594,0.0000
C01829=-24.227,95.023,39.203,178.2776,0.4750,0.0000
C01830=-21.221,93.510,39.027,177.6909,1.9849,0.0000
C01831=-19.458,91.164,38.697,178.4928,2.5231,0.0000
C01832=-18.041,88.518,38.031,-179.9182,-0.1571,0.0000
C01833=-16.662,86.143,37.169,-176.3239,-5.7975,0.0000
C01834=-15.030,84.409,36.333,-165.2581,-13.5086,0.0000
C01835=-12.558,83.543,35.726,-146.1515,-6.8803,0.0000
C01836=-8.530,83.594,35.484,-142.9367,2.3005,0.0000
C01837=-4.330,83.888,35.473,-142.7715,2.3885,0.0000
C01838=0.000,84.003,35.480,-142.7415,0.0004,0.0000
C01839=0.000,82.662,37.225,-142.2055,0.0004,0.0000
C01840=4.208,82.553,37.217,-142.2354,-2.4196,0.0000
C01841=8.324,82.270,37.229,-142.4103,-2.0928,0.0000
C01842=12.305,82.260,37.495,-146.1454,8.1058,0.0000
C01843=14.718,83.232,38.165,-167.2077,13.2282,0.0000
C01844=16.299,85.134,39.090,-177.2970,4.7574,0.0000
C01845=17.640,87.735,40.048,179.6311,-0.7865,0.0000
C01846=19.021,90.644,40.789,178.1721,-3.4318,0.0000
C01847=20.743,93.250,41.159,177.1705,-2.7402,0.0000
C01848=23.775,94.968,41.355,177.8447,-0.6817,0.0000
C01849=27.752,95.500,41.515,178.5424,0.0427,0.0000
C01850=31.992,94.679,41.678,179.9379,0.0198,0.0000
C01851=36.189,93.214,41.785,179.9917,0.0032,0.0000
C01852=40.323,91.502,41.785,179.9919,0.0036,0.0000
C01853=44.326,89.570,41.678,179.9421,0.0299,0.0000
C01854=47.905,87.153,41.515,178.9390,1.0006,0.0000
C01855=50.341,83.964,41.355,178.9574,2.0060,0.0000
C01856=51.270,80.606,41.159,179.9367,3.9353,0.0000
C01857=50.645,77.545,40.789,-178.8635,3.7173,0.0000
C01858=49.565,74.511,40.048,-179.7046,0.8170,0.0000
C01859=48.673,71.724,39.090,178.5413,-5.2696,0.0000
C01860=48.447,69.261,38.165,179.6754,-18.0958,0.0000
C01861=49.465,66.868,37.495,-159.5127,-29.9012,0.0000
C01862=52.288,64.059,37.229,-150.3090,-27.4069,0.0000
C01863=55.398,61.349,37.217,-149.9864,-27.3801,0.0000
C01864=58.451,58.451,37.225,-151.2608,-28.7396,0.0000
C01865=61.349,55.398,37.217,-152.6195,-30.0134,0.0000
C01866=64.059,52.288,37.229,-152.5923,-29.6900,0.0000
C01867=66.868,49.465,37.495,-150.0991,-20.4882,0.0000
C01868=69.261,48.447,38.165,-161.9042,0.3246,0.0000
C01869=71.724,48.673,39.090,-174.7304,1.4587,0.0000
C01870=74.511,49.565,40.048,179.1830,-0.2954,0.0000
C01871=77.545,50.645,40.789,176.2827,-1.1365,0.0000
C01872=80.606,51.270,41.159,176.0647,0.0633,0.0000
C01873=83.964,50.341,41.355,177.9940,1.0426,0.0000
